LIN {X 0,Y 195.72,Z 619.6,A -85,B 0,C 180,E1 -21671.148,E2 -21671.148} C_VEL
LIN {X 0,Y 194.07,Z 621.131,A -85,B 0,C 180,E1 -21673.162,E2 -21673.162} C_VEL
LIN {X 0,Y 191.846,Z 622.993,A -85,B 0,C 180,E1 -21677.306,E2 -21677.306} C_VEL
LIN {X 0,Y 190.603,Z 623.34,A -85,B 0,C 180,E1 -21681.521,E2 -21681.521} C_VEL
LIN {X 0,Y 190.275,Z 622.063,A -85,B 0,C 180,E1 -21685.766,E2 -21685.766} C_VEL
LIN {X 0,Y 190.318,Z 624.415,A -85,B 0,C 180,E1 -21690.003,E2 -21690.003} C_VEL
LIN {X 0,Y 190.137,Z 625.21,A -85,B 0,C 180,E1 -21693.626,E2 -21693.626} C_VEL
LIN {X 0,Y 190.28,Z 625.058,A -85,B 0,C 180,E1 -21696.364,E2 -21696.364} C_VEL
LIN {X 0,Y 191.05,Z 623.452,A -85,B 0,C 180,E1 -21700.601,E2 -21700.601} C_VEL
LIN {X 0,Y 192.667,Z 620.281,A -85,B 0,C 180,E1 -21704.797,E2 -21704.797} C_VEL
LIN {X 0,Y 194.637,Z 616.754,A -85,B 0,C 180,E1 -21707.876,E2 -21707.876} C_VEL
LIN {X 0,Y 197.217,Z 612.163,A -85,B 0,C 180,E1 -21710.879,E2 -21710.879} C_VEL
LIN {X 0,Y 200.069,Z 606.398,A -85,B 0,C 180,E1 -21713.83,E2 -21713.83} C_VEL
LIN {X 0,Y 203.568,Z 599.221,A -85,B 0,C 180,E1 -21716.67,E2 -21716.67} C_VEL
LIN {X 0,Y 207.615,Z 590.37,A -85,B 0,C 180,E1 -21719.398,E2 -21719.398} C_VEL
LIN {X 0,Y 211.864,Z 580.374,A -85,B 0,C 180,E1 -21721.779,E2 -21721.779} C_VEL
LIN {X 0,Y 215.55,Z 570.262,A -85,B 0,C 180,E1 -21723.664,E2 -21723.664} C_VEL
LIN {X 0,Y 219.069,Z 559.169,A -85,B 0,C 180,E1 -21725.275,E2 -21725.275} C_VEL
LIN {X 0,Y 222.34,Z 546.821,A -85,B 0,C 180,E1 -21726.631,E2 -21726.631} C_VEL
LIN {X 0,Y 225.036,Z 534.261,A -85,B 0,C 180,E1 -21727.59,E2 -21727.59} C_VEL
LIN {X 0,Y 227.03,Z 520.28,A -85,B 0,C 180,E1 -21728.346,E2 -21728.346} C_VEL
LIN {X 0,Y 230.459,Z 474.286,A -85,B 0,C 180,E1 -21729.931,E2 -21729.931} C_VEL
LIN {X 0,Y 230.155,Z 471.556,A -85,B 0,C 180,E1 -21730.175,E2 -21730.175} C_VEL
LIN {X 0,Y 225.508,Z 459.907,A -85,B 0,C 180,E1 -21732.317,E2 -21732.317} C_VEL
LIN {X 0,Y 220.788,Z 450.089,A -85,B 0,C 180,E1 -21734.626,E2 -21734.626} C_VEL
LIN {X 0,Y 216.678,Z 442.974,A -85,B 0,C 180,E1 -21736.78,E2 -21736.78} C_VEL
LIN {X 0,Y 214.755,Z 439.559,A -85,B 0,C 180,E1 -21737.912,E2 -21737.912} C_VEL
LIN {X 0,Y 211.682,Z 434.637,A -85,B 0,C 180,E1 -21739.814,E2 -21739.814} C_VEL
LIN {X 0,Y 208.202,Z 429.263,A -85,B 0,C 180,E1 -21742.258,E2 -21742.258} C_VEL
LIN {X 0,Y 204.808,Z 424.304,A -85,B 0,C 180,E1 -21745.032,E2 -21745.032} C_VEL
LIN {X 0,Y 203.656,Z 422.908,A -85,B 0,C 180,E1 -21746.097,E2 -21746.097} C_VEL
LIN {X 0,Y 199.168,Z 416.55,A -85,B 0,C 180,E1 -21751.575,E2 -21751.575} C_VEL
LIN {X 0,Y 196.529,Z 413.751,A -85,B 0,C 180,E1 -21757.393,E2 -21757.393} C_VEL
LIN {X 0,Y 196.055,Z 412.817,A -85,B 0,C 180,E1 -21761.178,E2 -21761.178} C_VEL
LIN {X 0,Y 196.746,Z 413.155,A -85,B 0,C 180,E1 -21765.52,E2 -21765.52} C_VEL
LIN {X 0,Y 198.963,Z 414.697,A -85,B 0,C 180,E1 -21770.26,E2 -21770.26} C_VEL
LIN {X 0,Y 201.05,Z 417.885,A -85,B 0,C 180,E1 -21773.351,E2 -21773.351} C_VEL
LIN {X 0,Y 204.042,Z 420.336,A -85,B 0,C 180,E1 -21776.378,E2 -21776.378} C_VEL
LIN {X 0,Y 206.331,Z 423.47,A -85,B 0,C 180,E1 -21778.445,E2 -21778.445} C_VEL
LIN {X 0,Y 208.258,Z 425.675,A -85,B 0,C 180,E1 -21779.91,E2 -21779.91} C_VEL
LIN {X 0,Y 211.756,Z 430.682,A -85,B 0,C 180,E1 -21782.378,E2 -21782.378} C_VEL
LIN {X 0,Y 215.572,Z 436.324,A -85,B 0,C 180,E1 -21784.701,E2 -21784.701} C_VEL
LIN {X 0,Y 220.508,Z 444.441,A -85,B 0,C 180,E1 -21787.367,E2 -21787.367} C_VEL
LIN {X 0,Y 225.524,Z 453.78,A -85,B 0,C 180,E1 -21789.803,E2 -21789.803} C_VEL
LIN {X 0,Y 229.635,Z 462.77,A -85,B 0,C 180,E1 -21791.651,E2 -21791.651} C_VEL
LIN {X 0,Y 231.003,Z 466.08,A -85,B 0,C 180,E1 -21792.254,E2 -21792.254} C_VEL
LIN {X 0,Y 227.309,Z 513.393,A -85,B 0,C 180,E1 -21793.884,E2 -21793.884} C_VEL
LIN {X 0,Y 225.489,Z 526.303,A -85,B 0,C 180,E1 -21794.616,E2 -21794.616} C_VEL
LIN {X 0,Y 223.106,Z 538.646,A -85,B 0,C 180,E1 -21795.645,E2 -21795.645} C_VEL
LIN {X 0,Y 220.057,Z 550.738,A -85,B 0,C 180,E1 -21797.031,E2 -21797.031} C_VEL
LIN {X 0,Y 216.86,Z 561.12,A -85,B 0,C 180,E1 -21798.567,E2 -21798.567} C_VEL
LIN {X 0,Y 213.017,Z 571.787,A -85,B 0,C 180,E1 -21800.579,E2 -21800.579} C_VEL
LIN {X 0,Y 208.985,Z 581.554,A -85,B 0,C 180,E1 -21802.981,E2 -21802.981} C_VEL
LIN {X 0,Y 204.885,Z 590.415,A -85,B 0,C 180,E1 -21805.78,E2 -21805.78} C_VEL
LIN {X 0,Y 201.513,Z 596.904,A -85,B 0,C 180,E1 -21808.382,E2 -21808.382} C_VEL
LIN {X 0,Y 198.132,Z 603.112,A -85,B 0,C 180,E1 -21811.641,E2 -21811.641} C_VEL
LIN {X 0,Y 195.241,Z 608.052,A -85,B 0,C 180,E1 -21815.166,E2 -21815.166} C_VEL
LIN {X 0,Y 193.362,Z 611.071,A -85,B 0,C 180,E1 -21818.162,E2 -21818.162} C_VEL
LIN {X 0,Y 191.904,Z 613.201,A -85,B 0,C 180,E1 -21821.24,E2 -21821.24} C_VEL
LIN {X 0,Y 190.5,Z 614.691,A -85,B 0,C 180,E1 -21825.493,E2 -21825.493} C_VEL
LIN {X 0,Y 189.985,Z 614.771,A -85,B 0,C 180,E1 -21828.248,E2 -21828.248} C_VEL
LIN {X 0,Y 189.755,Z 614.193,A -85,B 0,C 180,E1 -21831.059,E2 -21831.059} C_VEL
LIN {X 0,Y 189.779,Z 612.447,A -85,B 0,C 180,E1 -21834.56,E2 -21834.56} C_VEL
LIN {X 0,Y 190.323,Z 609.463,A -85,B 0,C 180,E1 -21838.138,E2 -21838.138} C_VEL
LIN {X 0,Y 191.202,Z 604.893,A -85,B 0,C 180,E1 -21841.906,E2 -21841.906} C_VEL
LIN {X 0,Y 192.232,Z 599.97,A -85,B 0,C 180,E1 -21844.948,E2 -21844.948} C_VEL
LIN {X 0,Y 193.763,Z 593.339,A -85,B 0,C 180,E1 -21848.172,E2 -21848.172} C_VEL
LIN {X 0,Y 195.561,Z 585.609,A -85,B 0,C 180,E1 -21851.126,E2 -21851.126} C_VEL
LIN {X 0,Y 197.618,Z 576.917,A -85,B 0,C 180,E1 -21853.785,E2 -21853.785} C_VEL
LIN {X 0,Y 199.933,Z 566.816,A -85,B 0,C 180,E1 -21856.255,E2 -21856.255} C_VEL
LIN {X 0,Y 201.923,Z 556.858,A -85,B 0,C 180,E1 -21858.198,E2 -21858.198} C_VEL
LIN {X 0,Y 204.183,Z 544.37,A -85,B 0,C 180,E1 -21860.088,E2 -21860.088} C_VEL
LIN {X 0,Y 205.884,Z 532.609,A -85,B 0,C 180,E1 -21861.445,E2 -21861.445} C_VEL
LIN {X 0,Y 207.28,Z 519.795,A -85,B 0,C 180,E1 -21862.512,E2 -21862.512} C_VEL
LIN {X 0,Y 208.32,Z 506.638,A -85,B 0,C 180,E1 -21863.215,E2 -21863.215} C_VEL
LIN {X 0,Y 211.141,Z 450.661,A -85,B 0,C 180,E1 -21865.247,E2 -21865.247} C_VEL
LIN {X 0,Y 202.81,Z 427.829,A -85,B 0,C 180,E1 -21867.418,E2 -21867.418} C_VEL
LIN {X 0,Y 193.596,Z 408.295,A -85,B 0,C 180,E1 -21869.803,E2 -21869.803} C_VEL
LIN {X 0,Y 193.445,Z 407.387,A -85,B 0,C 180,E1 -21869.932,E2 -21869.932} C_VEL
LIN {X 0,Y 192.983,Z 407.442,A -85,B 0,C 180,E1 -21874.174,E2 -21874.174} C_VEL
LIN {X 0,Y 193.081,Z 407.431,A -85,B 0,C 180,E1 -21878.369,E2 -21878.369} C_VEL
LIN {X 0,Y 192.854,Z 407.455,A -85,B 0,C 180,E1 -21882.627,E2 -21882.627} C_VEL
LIN {X 0,Y 192.758,Z 407.473,A -85,B 0,C 180,E1 -21886.956,E2 -21886.956} C_VEL
LIN {X 0,Y 192.636,Z 407.485,A -85,B 0,C 180,E1 -21891.394,E2 -21891.394} C_VEL
LIN {X 0,Y 192.663,Z 407.484,A -85,B 0,C 180,E1 -21894.222,E2 -21894.222} C_VEL
LIN {X 0,Y 192.642,Z 407.476,A -85,B 0,C 180,E1 -21898.886,E2 -21898.886} C_VEL
LIN {X 0,Y 192.59,Z 407.495,A -85,B 0,C 180,E1 -21904.442,E2 -21904.442} C_VEL
LIN {X 0,Y 192.647,Z 407.577,A -85,B 0,C 180,E1 -21905.627,E2 -21905.627} C_VEL
LIN {X 0,Y 200.514,Z 429.954,A -85,B 0,C 180,E1 -21907.562,E2 -21907.562} C_VEL
LIN {X 0,Y 204.611,Z 443.484,A -85,B 0,C 180,E1 -21908.602,E2 -21908.602} C_VEL
LIN {X 0,Y 200.833,Z 511.211,A -85,B 0,C 180,E1 -21911.922,E2 -21911.922} C_VEL
LIN {X 0,Y 199.882,Z 524.754,A -85,B 0,C 180,E1 -21912.963,E2 -21912.963} C_VEL
LIN {X 0,Y 198.418,Z 539.046,A -85,B 0,C 180,E1 -21914.534,E2 -21914.534} C_VEL
LIN {X 0,Y 196.966,Z 550.809,A -85,B 0,C 180,E1 -21916.264,E2 -21916.264} C_VEL
LIN {X 0,Y 195.299,Z 563.165,A -85,B 0,C 180,E1 -21918.585,E2 -21918.585} C_VEL
LIN {X 0,Y 193.693,Z 574.251,A -85,B 0,C 180,E1 -21921.251,E2 -21921.251} C_VEL
LIN {X 0,Y 192.55,Z 582.821,A -85,B 0,C 180,E1 -21923.791,E2 -21923.791} C_VEL
LIN {X 0,Y 191.558,Z 590.579,A -85,B 0,C 180,E1 -21926.61,E2 -21926.61} C_VEL
LIN {X 0,Y 190.673,Z 598.346,A -85,B 0,C 180,E1 -21930.159,E2 -21930.159} C_VEL
LIN {X 0,Y 190.126,Z 604.251,A -85,B 0,C 180,E1 -21933.667,E2 -21933.667} C_VEL
LIN {X 0,Y 189.785,Z 608.454,A -85,B 0,C 180,E1 -21936.992,E2 -21936.992} C_VEL
LIN {X 0,Y 189.845,Z 611.673,A -85,B 0,C 180,E1 -21940.538,E2 -21940.538} C_VEL
LIN {X 0,Y 190.37,Z 613.55,A -85,B 0,C 180,E1 -21943.699,E2 -21943.699} C_VEL
LIN {X 0,Y 191.399,Z 614.57,A -85,B 0,C 180,E1 -21947.272,E2 -21947.272} C_VEL
LIN {X 0,Y 192.6,Z 614.58,A -85,B 0,C 180,E1 -21950.122,E2 -21950.122} C_VEL
LIN {X 0,Y 194.924,Z 613.442,A -85,B 0,C 180,E1 -21953.79,E2 -21953.79} C_VEL
LIN {X 0,Y 197.152,Z 611.798,A -85,B 0,C 180,E1 -21956.445,E2 -21956.445} C_VEL
LIN {X 0,Y 200.801,Z 608.327,A -85,B 0,C 180,E1 -21960,E2 -21960} C_VEL
LIN {X 0,Y 205.018,Z 603.713,A -85,B 0,C 180,E1 -21963.203,E2 -21963.203} C_VEL
LIN {X 0,Y 209.825,Z 597.699,A -85,B 0,C 180,E1 -21966.249,E2 -21966.249} C_VEL
LIN {X 0,Y 214.647,Z 590.895,A -85,B 0,C 180,E1 -21968.853,E2 -21968.853} C_VEL
LIN {X 0,Y 220.368,Z 581.806,A -85,B 0,C 180,E1 -21971.497,E2 -21971.497} C_VEL
LIN {X 0,Y 225.068,Z 573.343,A -85,B 0,C 180,E1 -21973.423,E2 -21973.423} C_VEL
LIN {X 0,Y 230.657,Z 561.717,A -85,B 0,C 180,E1 -21975.462,E2 -21975.462} C_VEL
LIN {X 0,Y 235.084,Z 550.754,A -85,B 0,C 180,E1 -21976.939,E2 -21976.939} C_VEL
LIN {X 0,Y 239.295,Z 538.245,A -85,B 0,C 180,E1 -21978.24,E2 -21978.24} C_VEL
LIN {X 0,Y 242.468,Z 526.564,A -85,B 0,C 180,E1 -21979.141,E2 -21979.141} C_VEL
LIN {X 0,Y 245.063,Z 513.73,A -85,B 0,C 180,E1 -21979.856,E2 -21979.856} C_VEL
LIN {X 0,Y 249.279,Z 484.945,A -85,B 0,C 180,E1 -21981.013,E2 -21981.013} C_VEL
LIN {X 0,Y 249.307,Z 482.556,A -85,B 0,C 180,E1 -21981.299,E2 -21981.299} C_VEL
LIN {X 0,Y 248.726,Z 480.497,A -85,B 0,C 180,E1 -21981.926,E2 -21981.926} C_VEL
LIN {X 0,Y 247.718,Z 479.21,A -85,B 0,C 180,E1 -21982.755,E2 -21982.755} C_VEL
LIN {X 0,Y 244.844,Z 477.488,A -85,B 0,C 180,E1 -21985.136,E2 -21985.136} C_VEL
LIN {X 0,Y 244.529,Z 477.081,A -85,B 0,C 180,E1 -21985.474,E2 -21985.474} C_VEL
LIN {X 0,Y 243.393,Z 474.587,A -85,B 0,C 180,E1 -21987.16,E2 -21987.16} C_VEL
LIN {X 0,Y 242.23,Z 471.931,A -85,B 0,C 180,E1 -21989.553,E2 -21989.553} C_VEL
LIN {X 0,Y 241.395,Z 470.813,A -85,B 0,C 180,E1 -21992.407,E2 -21992.407} C_VEL
LIN {X 0,Y 241.409,Z 470.899,A -85,B 0,C 180,E1 -21995.609,E2 -21995.609} C_VEL
LIN {X 0,Y 242.353,Z 472.652,A -85,B 0,C 180,E1 -21998.736,E2 -21998.736} C_VEL
LIN {X 0,Y 243.872,Z 476.256,A -85,B 0,C 180,E1 -22001.516,E2 -22001.516} C_VEL
LIN {X 0,Y 245.796,Z 480.734,A -85,B 0,C 180,E1 -22003.961,E2 -22003.961} C_VEL
LIN {X 0,Y 246.892,Z 483.497,A -85,B 0,C 180,E1 -22005.123,E2 -22005.123} C_VEL
LIN {X 0,Y 240.741,Z 522.488,A -85,B 0,C 180,E1 -22006.758,E2 -22006.758} C_VEL
LIN {X 0,Y 237.486,Z 536.119,A -85,B 0,C 180,E1 -22007.542,E2 -22007.542} C_VEL
LIN {X 0,Y 233.407,Z 548.738,A -85,B 0,C 180,E1 -22008.518,E2 -22008.518} C_VEL
LIN {X 0,Y 228.53,Z 560.939,A -85,B 0,C 180,E1 -22009.777,E2 -22009.777} C_VEL
LIN {X 0,Y 222.432,Z 573.961,A -85,B 0,C 180,E1 -22011.682,E2 -22011.682} C_VEL
LIN {X 0,Y 217.63,Z 582.71,A -85,B 0,C 180,E1 -22013.318,E2 -22013.318} C_VEL
LIN {X 0,Y 211.65,Z 592.278,A -85,B 0,C 180,E1 -22015.636,E2 -22015.636} C_VEL
LIN {X 0,Y 206.176,Z 600.165,A -85,B 0,C 180,E1 -22018.109,E2 -22018.109} C_VEL
LIN {X 0,Y 200.984,Z 607.02,A -85,B 0,C 180,E1 -22020.95,E2 -22020.95} C_VEL
LIN {X 0,Y 196.912,Z 611.796,A -85,B 0,C 180,E1 -22023.507,E2 -22023.507} C_VEL
LIN {X 0,Y 193.283,Z 615.915,A -85,B 0,C 180,E1 -22026.427,E2 -22026.427} C_VEL
LIN {X 0,Y 191.042,Z 618.136,A -85,B 0,C 180,E1 -22028.418,E2 -22028.418} C_VEL
LIN {X 0,Y 187.282,Z 621.302,A -85,B 0,C 180,E1 -22032.533,E2 -22032.533} C_VEL
LIN {X 0,Y 184.903,Z 622.943,A -85,B 0,C 180,E1 -22036.82,E2 -22036.82} C_VEL
LIN {X 0,Y 183.563,Z 622.993,A -85,B 0,C 180,E1 -22041.194,E2 -22041.194} C_VEL
LIN {X 0,Y 183.201,Z 621.563,A -85,B 0,C 180,E1 -22045.722,E2 -22045.722} C_VEL
LIN {X 0,Y 183.116,Z 623.011,A -85,B 0,C 180,E1 -22047.803,E2 -22047.803} C_VEL
LIN {X 0,Y 183.22,Z 624.102,A -85,B 0,C 180,E1 -22050.003,E2 -22050.003} C_VEL
LIN {X 0,Y 183.054,Z 624.966,A -85,B 0,C 180,E1 -22053.417,E2 -22053.417} C_VEL
LIN {X 0,Y 183.213,Z 624.889,A -85,B 0,C 180,E1 -22056.611,E2 -22056.611} C_VEL
LIN {X 0,Y 183.517,Z 624.357,A -85,B 0,C 180,E1 -22058.814,E2 -22058.814} C_VEL
LIN {X 0,Y 184.817,Z 622.081,A -85,B 0,C 180,E1 -22063.192,E2 -22063.192} C_VEL
LIN {X 0,Y 186.415,Z 619.31,A -85,B 0,C 180,E1 -22066.428,E2 -22066.428} C_VEL
LIN {X 0,Y 188.727,Z 615.542,A -85,B 0,C 180,E1 -22069.585,E2 -22069.585} C_VEL
LIN {X 0,Y 191.568,Z 610.685,A -85,B 0,C 180,E1 -22072.659,E2 -22072.659} C_VEL
LIN {X 0,Y 195.358,Z 603.525,A -85,B 0,C 180,E1 -22076.151,E2 -22076.151} C_VEL
LIN {X 0,Y 199.338,Z 595.77,A -85,B 0,C 180,E1 -22079.001,E2 -22079.001} C_VEL
LIN {X 0,Y 203.05,Z 587.911,A -85,B 0,C 180,E1 -22081.28,E2 -22081.28} C_VEL
LIN {X 0,Y 207.593,Z 577.326,A -85,B 0,C 180,E1 -22083.67,E2 -22083.67} C_VEL
LIN {X 0,Y 211.547,Z 566.614,A -85,B 0,C 180,E1 -22085.551,E2 -22085.551} C_VEL
LIN {X 0,Y 215.332,Z 554.54,A -85,B 0,C 180,E1 -22087.145,E2 -22087.145} C_VEL
LIN {X 0,Y 218.326,Z 542.986,A -85,B 0,C 180,E1 -22088.294,E2 -22088.294} C_VEL
LIN {X 0,Y 220.995,Z 529.936,A -85,B 0,C 180,E1 -22089.205,E2 -22089.205} C_VEL
LIN {X 0,Y 222.7,Z 516.089,A -85,B 0,C 180,E1 -22089.872,E2 -22089.872} C_VEL
LIN {X 0,Y 225.877,Z 475.392,A -85,B 0,C 180,E1 -22091.274,E2 -22091.274} C_VEL
LIN {X 0,Y 222.659,Z 466.731,A -85,B 0,C 180,E1 -22092.857,E2 -22092.857} C_VEL
LIN {X 0,Y 218.886,Z 458.171,A -85,B 0,C 180,E1 -22094.81,E2 -22094.81} C_VEL
LIN {X 0,Y 214.768,Z 450.261,A -85,B 0,C 180,E1 -22097.072,E2 -22097.072} C_VEL
LIN {X 0,Y 211.767,Z 444.948,A -85,B 0,C 180,E1 -22098.91,E2 -22098.91} C_VEL
LIN {X 0,Y 209.193,Z 440.674,A -85,B 0,C 180,E1 -22100.6,E2 -22100.6} C_VEL
LIN {X 0,Y 205.948,Z 435.399,A -85,B 0,C 180,E1 -22103.058,E2 -22103.058} C_VEL
LIN {X 0,Y 202.382,Z 429.965,A -85,B 0,C 180,E1 -22106.246,E2 -22106.246} C_VEL
LIN {X 0,Y 197.854,Z 423.395,A -85,B 0,C 180,E1 -22111.935,E2 -22111.935} C_VEL
LIN {X 0,Y 195.378,Z 420.67,A -85,B 0,C 180,E1 -22117.809,E2 -22117.809} C_VEL
LIN {X 0,Y 195.019,Z 419.868,A -85,B 0,C 180,E1 -22121.075,E2 -22121.075} C_VEL
LIN {X 0,Y 195.667,Z 420.166,A -85,B 0,C 180,E1 -22125.438,E2 -22125.438} C_VEL
LIN {X 0,Y 197.663,Z 421.666,A -85,B 0,C 180,E1 -22129.925,E2 -22129.925} C_VEL
LIN {X 0,Y 199.777,Z 424.81,A -85,B 0,C 180,E1 -22133.118,E2 -22133.118} C_VEL
LIN {X 0,Y 202.528,Z 427.29,A -85,B 0,C 180,E1 -22136.02,E2 -22136.02} C_VEL
LIN {X 0,Y 204.674,Z 430.212,A -85,B 0,C 180,E1 -22138.032,E2 -22138.032} C_VEL
LIN {X 0,Y 206.217,Z 432.116,A -85,B 0,C 180,E1 -22139.268,E2 -22139.268} C_VEL
LIN {X 0,Y 210.405,Z 438.444,A -85,B 0,C 180,E1 -22142.342,E2 -22142.342} C_VEL
LIN {X 0,Y 213.122,Z 442.572,A -85,B 0,C 180,E1 -22144.044,E2 -22144.044} C_VEL
LIN {X 0,Y 217.554,Z 450.264,A -85,B 0,C 180,E1 -22146.598,E2 -22146.598} C_VEL
LIN {X 0,Y 222.038,Z 458.885,A -85,B 0,C 180,E1 -22148.908,E2 -22148.908} C_VEL
LIN {X 0,Y 225.885,Z 467.674,A -85,B 0,C 180,E1 -22150.759,E2 -22150.759} C_VEL
LIN {X 0,Y 226.279,Z 468.651,A -85,B 0,C 180,E1 -22150.944,E2 -22150.944} C_VEL
LIN {X 0,Y 222.592,Z 513.888,A -85,B 0,C 180,E1 -22152.537,E2 -22152.537} C_VEL
LIN {X 0,Y 220.629,Z 527.039,A -85,B 0,C 180,E1 -22153.3,E2 -22153.3} C_VEL
LIN {X 0,Y 218.1,Z 539.38,A -85,B 0,C 180,E1 -22154.36,E2 -22154.36} C_VEL
LIN {X 0,Y 214.947,Z 551.16,A -85,B 0,C 180,E1 -22155.734,E2 -22155.734} C_VEL
LIN {X 0,Y 211.331,Z 562.279,A -85,B 0,C 180,E1 -22157.416,E2 -22157.416} C_VEL
LIN {X 0,Y 207.656,Z 571.974,A -85,B 0,C 180,E1 -22159.29,E2 -22159.29} C_VEL
LIN {X 0,Y 203.87,Z 580.756,A -85,B 0,C 180,E1 -22161.439,E2 -22161.439} C_VEL
LIN {X 0,Y 199.436,Z 589.861,A -85,B 0,C 180,E1 -22164.303,E2 -22164.303} C_VEL
LIN {X 0,Y 195.34,Z 597.352,A -85,B 0,C 180,E1 -22167.354,E2 -22167.354} C_VEL
LIN {X 0,Y 191.526,Z 603.807,A -85,B 0,C 180,E1 -22170.913,E2 -22170.913} C_VEL
LIN {X 0,Y 188.954,Z 607.901,A -85,B 0,C 180,E1 -22173.912,E2 -22173.912} C_VEL
LIN {X 0,Y 186.464,Z 611.57,A -85,B 0,C 180,E1 -22177.669,E2 -22177.669} C_VEL
LIN {X 0,Y 185.053,Z 613.449,A -85,B 0,C 180,E1 -22180.57,E2 -22180.57} C_VEL
LIN {X 0,Y 183.974,Z 614.608,A -85,B 0,C 180,E1 -22183.459,E2 -22183.459} C_VEL
LIN {X 0,Y 183.118,Z 615.045,A -85,B 0,C 180,E1 -22186.821,E2 -22186.821} C_VEL
LIN {X 0,Y 182.676,Z 614.523,A -85,B 0,C 180,E1 -22190.305,E2 -22190.305} C_VEL
LIN {X 0,Y 182.65,Z 612.938,A -85,B 0,C 180,E1 -22193.905,E2 -22193.905} C_VEL
LIN {X 0,Y 183.127,Z 610.142,A -85,B 0,C 180,E1 -22197.599,E2 -22197.599} C_VEL
LIN {X 0,Y 183.983,Z 605.786,A -85,B 0,C 180,E1 -22201.473,E2 -22201.473} C_VEL
LIN {X 0,Y 185.24,Z 599.853,A -85,B 0,C 180,E1 -22205.33,E2 -22205.33} C_VEL
LIN {X 0,Y 186.949,Z 592.733,A -85,B 0,C 180,E1 -22208.832,E2 -22208.832} C_VEL
LIN {X 0,Y 189.024,Z 584.112,A -85,B 0,C 180,E1 -22212.134,E2 -22212.134} C_VEL
LIN {X 0,Y 191.037,Z 575.886,A -85,B 0,C 180,E1 -22214.646,E2 -22214.646} C_VEL
LIN {X 0,Y 193.444,Z 565.663,A -85,B 0,C 180,E1 -22217.14,E2 -22217.14} C_VEL
LIN {X 0,Y 195.832,Z 553.864,A -85,B 0,C 180,E1 -22219.399,E2 -22219.399} C_VEL
LIN {X 0,Y 197.9,Z 542.431,A -85,B 0,C 180,E1 -22221.086,E2 -22221.086} C_VEL
LIN {X 0,Y 199.76,Z 529.153,A -85,B 0,C 180,E1 -22222.543,E2 -22222.543} C_VEL
LIN {X 0,Y 201.13,Z 516.229,A -85,B 0,C 180,E1 -22223.54,E2 -22223.54} C_VEL
LIN {X 0,Y 202.134,Z 501.041,A -85,B 0,C 180,E1 -22224.239,E2 -22224.239} C_VEL
LIN {X 0,Y 204.656,Z 452.16,A -85,B 0,C 180,E1 -22226.059,E2 -22226.059} C_VEL
LIN {X 0,Y 196.883,Z 430.644,A -85,B 0,C 180,E1 -22228.2,E2 -22228.2} C_VEL
LIN {X 0,Y 187.869,Z 411.874,A -85,B 0,C 180,E1 -22230.62,E2 -22230.62} C_VEL
LIN {X 0,Y 186.468,Z 409.162,A -85,B 0,C 180,E1 -22231.009,E2 -22231.009} C_VEL
LIN {X 0,Y 186.288,Z 408.284,A -85,B 0,C 180,E1 -22231.145,E2 -22231.145} C_VEL
LIN {X 0,Y 186.031,Z 408.312,A -85,B 0,C 180,E1 -22238.689,E2 -22238.689} C_VEL
LIN {X 0,Y 185.766,Z 408.338,A -85,B 0,C 180,E1 -22243.117,E2 -22243.117} C_VEL
LIN {X 0,Y 185.69,Z 408.349,A -85,B 0,C 180,E1 -22247.622,E2 -22247.622} C_VEL
LIN {X 0,Y 185.596,Z 408.367,A -85,B 0,C 180,E1 -22252.248,E2 -22252.248} C_VEL
LIN {X 0,Y 185.558,Z 408.353,A -85,B 0,C 180,E1 -22257.029,E2 -22257.029} C_VEL
LIN {X 0,Y 185.575,Z 408.357,A -85,B 0,C 180,E1 -22259.49,E2 -22259.49} C_VEL
LIN {X 0,Y 185.568,Z 408.369,A -85,B 0,C 180,E1 -22264.944,E2 -22264.944} C_VEL
LIN {X 0,Y 193.936,Z 432.102,A -85,B 0,C 180,E1 -22267.116,E2 -22267.116} C_VEL
LIN {X 0,Y 197.668,Z 444.58,A -85,B 0,C 180,E1 -22268.114,E2 -22268.114} C_VEL
LIN {X 0,Y 193.894,Z 511.321,A -85,B 0,C 180,E1 -22271.52,E2 -22271.52} C_VEL
LIN {X 0,Y 193.005,Z 523.779,A -85,B 0,C 180,E1 -22272.491,E2 -22272.491} C_VEL
LIN {X 0,Y 191.681,Z 536.813,A -85,B 0,C 180,E1 -22273.921,E2 -22273.921} C_VEL
LIN {X 0,Y 190.13,Z 549.47,A -85,B 0,C 180,E1 -22275.757,E2 -22275.757} C_VEL
LIN {X 0,Y 188.605,Z 560.762,A -85,B 0,C 180,E1 -22277.876,E2 -22277.876} C_VEL
LIN {X 0,Y 187.067,Z 571.191,A -85,B 0,C 180,E1 -22280.306,E2 -22280.306} C_VEL
LIN {X 0,Y 185.815,Z 579.758,A -85,B 0,C 180,E1 -22282.759,E2 -22282.759} C_VEL
LIN {X 0,Y 184.702,Z 588.168,A -85,B 0,C 180,E1 -22285.725,E2 -22285.725} C_VEL
LIN {X 0,Y 183.82,Z 595.508,A -85,B 0,C 180,E1 -22288.926,E2 -22288.926} C_VEL
LIN {X 0,Y 183.333,Z 600.917,A -85,B 0,C 180,E1 -22291.841,E2 -22291.841} C_VEL
LIN {X 0,Y 182.866,Z 605.595,A -85,B 0,C 180,E1 -22294.991,E2 -22294.991} C_VEL
LIN {X 0,Y 182.685,Z 609.658,A -85,B 0,C 180,E1 -22298.577,E2 -22298.577} C_VEL
LIN {X 0,Y 182.938,Z 612.464,A -85,B 0,C 180,E1 -22302.101,E2 -22302.101} C_VEL
LIN {X 0,Y 183.426,Z 613.712,A -85,B 0,C 180,E1 -22304.442,E2 -22304.442} C_VEL
LIN {X 0,Y 184.067,Z 614.506,A -85,B 0,C 180,E1 -22306.756,E2 -22306.756} C_VEL
LIN {X 0,Y 185.463,Z 614.885,A -85,B 0,C 180,E1 -22310.128,E2 -22310.128} C_VEL
LIN {X 0,Y 187.522,Z 614.276,A -85,B 0,C 180,E1 -22313.544,E2 -22313.544} C_VEL
LIN {X 0,Y 190.065,Z 612.795,A -85,B 0,C 180,E1 -22316.676,E2 -22316.676} C_VEL
LIN {X 0,Y 193.425,Z 610.128,A -85,B 0,C 180,E1 -22320,E2 -22320} C_VEL
LIN {X 0,Y 197.023,Z 606.736,A -85,B 0,C 180,E1 -22322.884,E2 -22322.884} C_VEL
LIN {X 0,Y 201.792,Z 601.674,A -85,B 0,C 180,E1 -22325.997,E2 -22325.997} C_VEL
LIN {X 0,Y 206.702,Z 595.648,A -85,B 0,C 180,E1 -22328.773,E2 -22328.773} C_VEL
LIN {X 0,Y 212.355,Z 587.929,A -85,B 0,C 180,E1 -22331.453,E2 -22331.453} C_VEL
LIN {X 0,Y 218.267,Z 578.607,A -85,B 0,C 180,E1 -22333.937,E2 -22333.937} C_VEL
LIN {X 0,Y 223.827,Z 568.571,A -85,B 0,C 180,E1 -22335.947,E2 -22335.947} C_VEL
LIN {X 0,Y 228.969,Z 557.747,A -85,B 0,C 180,E1 -22337.656,E2 -22337.656} C_VEL
LIN {X 0,Y 233.721,Z 545.754,A -85,B 0,C 180,E1 -22339.099,E2 -22339.099} C_VEL
LIN {X 0,Y 238.001,Z 532.294,A -85,B 0,C 180,E1 -22340.302,E2 -22340.302} C_VEL
LIN {X 0,Y 241.53,Z 517.671,A -85,B 0,C 180,E1 -22341.216,E2 -22341.216} C_VEL
LIN {X 0,Y 246.734,Z 484.983,A -85,B 0,C 180,E1 -22342.551,E2 -22342.551} C_VEL
LIN {X 0,Y 246.958,Z 483.027,A -85,B 0,C 180,E1 -22342.679,E2 -22342.679} C_VEL
LIN {X 0,Y 245.435,Z 479.266,A -85,B 0,C 180,E1 -22344.338,E2 -22344.338} C_VEL
LIN {X 0,Y 244.529,Z 477.081,A -85,B 0,C 180,E1 -22345.474,E2 -22345.474} C_VEL
LIN {X 0,Y 243.399,Z 476.014,A -85,B 0,C 180,E1 -22346.816,E2 -22346.816} C_VEL
LIN {X 0,Y 242.248,Z 476.015,A -85,B 0,C 180,E1 -22348.196,E2 -22348.196} C_VEL
LIN {X 0,Y 240.077,Z 477.675,A -85,B 0,C 180,E1 -22351.973,E2 -22351.973} C_VEL
LIN {X 0,Y 239.872,Z 477.7,A -85,B 0,C 180,E1 -22352.935,E2 -22352.935} C_VEL
LIN {X 0,Y 240.01,Z 478.093,A -85,B 0,C 180,E1 -22356.08,E2 -22356.08} C_VEL
LIN {X 0,Y 240.713,Z 479.367,A -85,B 0,C 180,E1 -22358.334,E2 -22358.334} C_VEL
LIN {X 0,Y 242.003,Z 482.826,A -85,B 0,C 180,E1 -22361.043,E2 -22361.043} C_VEL
LIN {X 0,Y 243.655,Z 486.99,A -85,B 0,C 180,E1 -22363.356,E2 -22363.356} C_VEL
LIN {X 0,Y 243.924,Z 488.048,A -85,B 0,C 180,E1 -22363.749,E2 -22363.749} C_VEL
LIN {X 0,Y 238.424,Z 521.478,A -85,B 0,C 180,E1 -22365.119,E2 -22365.119} C_VEL
LIN {X 0,Y 235.029,Z 535.099,A -85,B 0,C 180,E1 -22365.87,E2 -22365.87} C_VEL
LIN {X 0,Y 230.905,Z 547.469,A -85,B 0,C 180,E1 -22366.782,E2 -22366.782} C_VEL
LIN {X 0,Y 225.857,Z 559.813,A -85,B 0,C 180,E1 -22368.012,E2 -22368.012} C_VEL
LIN {X 0,Y 220.571,Z 570.831,A -85,B 0,C 180,E1 -22369.522,E2 -22369.522} C_VEL
LIN {X 0,Y 214.342,Z 581.763,A -85,B 0,C 180,E1 -22371.469,E2 -22371.469} C_VEL
LIN {X 0,Y 208.005,Z 591.495,A -85,B 0,C 180,E1 -22373.755,E2 -22373.755} C_VEL
LIN {X 0,Y 202.149,Z 599.406,A -85,B 0,C 180,E1 -22376.206,E2 -22376.206} C_VEL
LIN {X 0,Y 196.877,Z 605.88,A -85,B 0,C 180,E1 -22378.831,E2 -22378.831} C_VEL
LIN {X 0,Y 192.002,Z 611.19,A -85,B 0,C 180,E1 -22381.589,E2 -22381.589} C_VEL
LIN {X 0,Y 188.043,Z 615.342,A -85,B 0,C 180,E1 -22384.548,E2 -22384.548} C_VEL
LIN {X 0,Y 184.485,Z 618.568,A -85,B 0,C 180,E1 -22387.611,E2 -22387.611} C_VEL
LIN {X 0,Y 180.523,Z 621.485,A -85,B 0,C 180,E1 -22391.857,E2 -22391.857} C_VEL
LIN {X 0,Y 177.981,Z 622.803,A -85,B 0,C 180,E1 -22396.298,E2 -22396.298} C_VEL
LIN {X 0,Y 176.545,Z 622.635,A -85,B 0,C 180,E1 -22400.841,E2 -22400.841} C_VEL
LIN {X 0,Y 176.138,Z 621.012,A -85,B 0,C 180,E1 -22405.426,E2 -22405.426} C_VEL
LIN {X 0,Y 176.023,Z 622.601,A -85,B 0,C 180,E1 -22407.715,E2 -22407.715} C_VEL
LIN {X 0,Y 176.124,Z 623.774,A -85,B 0,C 180,E1 -22410.003,E2 -22410.003} C_VEL
LIN {X 0,Y 175.971,Z 624.644,A -85,B 0,C 180,E1 -22413.178,E2 -22413.178} C_VEL
LIN {X 0,Y 176.142,Z 624.708,A -85,B 0,C 180,E1 -22416.878,E2 -22416.878} C_VEL
LIN {X 0,Y 176.481,Z 624.25,A -85,B 0,C 180,E1 -22419.169,E2 -22419.169} C_VEL
LIN {X 0,Y 177.066,Z 623.377,A -85,B 0,C 180,E1 -22421.45,E2 -22421.45} C_VEL
LIN {X 0,Y 178.917,Z 620.417,A -85,B 0,C 180,E1 -22425.963,E2 -22425.963} C_VEL
LIN {X 0,Y 181.175,Z 617.099,A -85,B 0,C 180,E1 -22429.255,E2 -22429.255} C_VEL
LIN {X 0,Y 183.995,Z 612.754,A -85,B 0,C 180,E1 -22432.458,E2 -22432.458} C_VEL
LIN {X 0,Y 187.784,Z 606.289,A -85,B 0,C 180,E1 -22436.074,E2 -22436.074} C_VEL
LIN {X 0,Y 191.723,Z 599.201,A -85,B 0,C 180,E1 -22439.062,E2 -22439.062} C_VEL
LIN {X 0,Y 196.214,Z 590.453,A -85,B 0,C 180,E1 -22441.895,E2 -22441.895} C_VEL
LIN {X 0,Y 200.488,Z 581.56,A -85,B 0,C 180,E1 -22444.119,E2 -22444.119} C_VEL
LIN {X 0,Y 204.504,Z 571.905,A -85,B 0,C 180,E1 -22446.055,E2 -22446.055} C_VEL
LIN {X 0,Y 208.31,Z 561.384,A -85,B 0,C 180,E1 -22447.701,E2 -22447.701} C_VEL
LIN {X 0,Y 211.85,Z 549.762,A -85,B 0,C 180,E1 -22449.076,E2 -22449.076} C_VEL
LIN {X 0,Y 214.793,Z 537.91,A -85,B 0,C 180,E1 -22450.106,E2 -22450.106} C_VEL
LIN {X 0,Y 217.24,Z 524.497,A -85,B 0,C 180,E1 -22450.925,E2 -22450.925} C_VEL
LIN {X 0,Y 218.876,Z 507.47,A -85,B 0,C 180,E1 -22451.614,E2 -22451.614} C_VEL
LIN {X 0,Y 221.346,Z 477.75,A -85,B 0,C 180,E1 -22452.621,E2 -22452.621} C_VEL
LIN {X 0,Y 217.326,Z 467.199,A -85,B 0,C 180,E1 -22454.8,E2 -22454.8} C_VEL
LIN {X 0,Y 213.819,Z 459.719,A -85,B 0,C 180,E1 -22456.775,E2 -22456.775} C_VEL
LIN {X 0,Y 209.792,Z 451.786,A -85,B 0,C 180,E1 -22459.325,E2 -22459.325} C_VEL
LIN {X 0,Y 206.719,Z 446.565,A -85,B 0,C 180,E1 -22461.472,E2 -22461.472} C_VEL
LIN {X 0,Y 203.846,Z 441.711,A -85,B 0,C 180,E1 -22463.774,E2 -22463.774} C_VEL
LIN {X 0,Y 200.529,Z 436.382,A -85,B 0,C 180,E1 -22466.969,E2 -22466.969} C_VEL
LIN {X 0,Y 196.543,Z 430.276,A -85,B 0,C 180,E1 -22472.299,E2 -22472.299} C_VEL
LIN {X 0,Y 194.244,Z 427.581,A -85,B 0,C 180,E1 -22478.232,E2 -22478.232} C_VEL
LIN {X 0,Y 193.983,Z 426.919,A -85,B 0,C 180,E1 -22480.97,E2 -22480.97} C_VEL
LIN {X 0,Y 194.592,Z 427.156,A -85,B 0,C 180,E1 -22485.356,E2 -22485.356} C_VEL
LIN {X 0,Y 196.366,Z 428.6,A -85,B 0,C 180,E1 -22489.561,E2 -22489.561} C_VEL
LIN {X 0,Y 198.487,Z 431.752,A -85,B 0,C 180,E1 -22492.862,E2 -22492.862} C_VEL
LIN {X 0,Y 200.825,Z 433.945,A -85,B 0,C 180,E1 -22495.453,E2 -22495.453} C_VEL
LIN {X 0,Y 203.119,Z 437.021,A -85,B 0,C 180,E1 -22497.675,E2 -22497.675} C_VEL
LIN {X 0,Y 204.188,Z 438.572,A -85,B 0,C 180,E1 -22498.613,E2 -22498.613} C_VEL
LIN {X 0,Y 208.166,Z 444.784,A -85,B 0,C 180,E1 -22501.685,E2 -22501.685} C_VEL
LIN {X 0,Y 210.592,Z 448.667,A -85,B 0,C 180,E1 -22503.306,E2 -22503.306} C_VEL
LIN {X 0,Y 215.21,Z 457.057,A -85,B 0,C 180,E1 -22506.119,E2 -22506.119} C_VEL
LIN {X 0,Y 219.303,Z 465.515,A -85,B 0,C 180,E1 -22508.332,E2 -22508.332} C_VEL
LIN {X 0,Y 221.751,Z 471.416,A -85,B 0,C 180,E1 -22509.615,E2 -22509.615} C_VEL
LIN {X 0,Y 218.076,Z 514.012,A -85,B 0,C 180,E1 -22511.111,E2 -22511.111} C_VEL
LIN {X 0,Y 216.062,Z 527.07,A -85,B 0,C 180,E1 -22511.869,E2 -22511.869} C_VEL
LIN {X 0,Y 213.644,Z 538.53,A -85,B 0,C 180,E1 -22512.839,E2 -22512.839} C_VEL
LIN {X 0,Y 210.636,Z 549.617,A -85,B 0,C 180,E1 -22514.083,E2 -22514.083} C_VEL
LIN {X 0,Y 206.831,Z 561.032,A -85,B 0,C 180,E1 -22515.774,E2 -22515.774} C_VEL
LIN {X 0,Y 202.8,Z 571.296,A -85,B 0,C 180,E1 -22517.736,E2 -22517.736} C_VEL
LIN {X 0,Y 198.617,Z 580.501,A -85,B 0,C 180,E1 -22519.97,E2 -22519.97} C_VEL
LIN {X 0,Y 194.37,Z 588.9,A -85,B 0,C 180,E1 -22522.598,E2 -22522.598} C_VEL
LIN {X 0,Y 190.482,Z 595.762,A -85,B 0,C 180,E1 -22525.315,E2 -22525.315} C_VEL
LIN {X 0,Y 186.384,Z 602.4,A -85,B 0,C 180,E1 -22528.75,E2 -22528.75} C_VEL
LIN {X 0,Y 182.715,Z 607.798,A -85,B 0,C 180,E1 -22532.582,E2 -22532.582} C_VEL
LIN {X 0,Y 180.449,Z 610.985,A -85,B 0,C 180,E1 -22535.748,E2 -22535.748} C_VEL
LIN {X 0,Y 178.584,Z 613.287,A -85,B 0,C 180,E1 -22539.026,E2 -22539.026} C_VEL
LIN {X 0,Y 177.182,Z 614.705,A -85,B 0,C 180,E1 -22542.401,E2 -22542.401} C_VEL
LIN {X 0,Y 176.191,Z 615.239,A -85,B 0,C 180,E1 -22545.889,E2 -22545.889} C_VEL
LIN {X 0,Y 175.591,Z 614.659,A -85,B 0,C 180,E1 -22550.175,E2 -22550.175} C_VEL
LIN {X 0,Y 175.522,Z 613.367,A -85,B 0,C 180,E1 -22553.208,E2 -22553.208} C_VEL
LIN {X 0,Y 175.907,Z 610.729,A -85,B 0,C 180,E1 -22557.036,E2 -22557.036} C_VEL
LIN {X 0,Y 176.73,Z 606.628,A -85,B 0,C 180,E1 -22561.03,E2 -22561.03} C_VEL
LIN {X 0,Y 177.697,Z 602.242,A -85,B 0,C 180,E1 -22564.208,E2 -22564.208} C_VEL
LIN {X 0,Y 179.045,Z 596.475,A -85,B 0,C 180,E1 -22567.495,E2 -22567.495} C_VEL
LIN {X 0,Y 180.822,Z 589.363,A -85,B 0,C 180,E1 -22570.706,E2 -22570.706} C_VEL
LIN {X 0,Y 183.005,Z 580.865,A -85,B 0,C 180,E1 -22573.758,E2 -22573.758} C_VEL
LIN {X 0,Y 185.474,Z 570.969,A -85,B 0,C 180,E1 -22576.577,E2 -22576.577} C_VEL
LIN {X 0,Y 187.946,Z 559.997,A -85,B 0,C 180,E1 -22579.017,E2 -22579.017} C_VEL
LIN {X 0,Y 190.204,Z 548.836,A -85,B 0,C 180,E1 -22580.962,E2 -22580.962} C_VEL
LIN {X 0,Y 192.219,Z 536.665,A -85,B 0,C 180,E1 -22582.59,E2 -22582.59} C_VEL
LIN {X 0,Y 193.92,Z 522.967,A -85,B 0,C 180,E1 -22583.919,E2 -22583.919} C_VEL
LIN {X 0,Y 195.234,Z 509.783,A -85,B 0,C 180,E1 -22584.737,E2 -22584.737} C_VEL
LIN {X 0,Y 198.236,Z 453.578,A -85,B 0,C 180,E1 -22586.925,E2 -22586.925} C_VEL
LIN {X 0,Y 190.875,Z 433.359,A -85,B 0,C 180,E1 -22589.039,E2 -22589.039} C_VEL
LIN {X 0,Y 182.601,Z 416.1,A -85,B 0,C 180,E1 -22591.36,E2 -22591.36} C_VEL
LIN {X 0,Y 179.379,Z 410.332,A -85,B 0,C 180,E1 -22592.278,E2 -22592.278} C_VEL
LIN {X 0,Y 179.108,Z 409.17,A -85,B 0,C 180,E1 -22592.457,E2 -22592.457} C_VEL
LIN {X 0,Y 178.98,Z 409.192,A -85,B 0,C 180,E1 -22599.034,E2 -22599.034} C_VEL
LIN {X 0,Y 178.688,Z 409.222,A -85,B 0,C 180,E1 -22603.647,E2 -22603.647} C_VEL
LIN {X 0,Y 178.65,Z 409.221,A -85,B 0,C 180,E1 -22608.34,E2 -22608.34} C_VEL
LIN {X 0,Y 178.51,Z 409.249,A -85,B 0,C 180,E1 -22613.182,E2 -22613.182} C_VEL
LIN {X 0,Y 178.483,Z 409.233,A -85,B 0,C 180,E1 -22618.194,E2 -22618.194} C_VEL
LIN {X 0,Y 178.474,Z 409.249,A -85,B 0,C 180,E1 -22620.788,E2 -22620.788} C_VEL
LIN {X 0,Y 178.515,Z 409.284,A -85,B 0,C 180,E1 -22624.291,E2 -22624.291} C_VEL
LIN {X 0,Y 187.333,Z 434.221,A -85,B 0,C 180,E1 -22626.633,E2 -22626.633} C_VEL
LIN {X 0,Y 190.778,Z 445.645,A -85,B 0,C 180,E1 -22627.597,E2 -22627.597} C_VEL
LIN {X 0,Y 186.946,Z 511.516,A -85,B 0,C 180,E1 -22631.093,E2 -22631.093} C_VEL
LIN {X 0,Y 185.888,Z 525.026,A -85,B 0,C 180,E1 -22632.202,E2 -22632.202} C_VEL
LIN {X 0,Y 184.449,Z 538.717,A -85,B 0,C 180,E1 -22633.815,E2 -22633.815} C_VEL
LIN {X 0,Y 182.82,Z 551.474,A -85,B 0,C 180,E1 -22635.832,E2 -22635.832} C_VEL
LIN {X 0,Y 181.17,Z 563.081,A -85,B 0,C 180,E1 -22638.182,E2 -22638.182} C_VEL
LIN {X 0,Y 179.589,Z 573.584,A -85,B 0,C 180,E1 -22640.873,E2 -22640.873} C_VEL
LIN {X 0,Y 178.333,Z 582.722,A -85,B 0,C 180,E1 -22643.762,E2 -22643.762} C_VEL
LIN {X 0,Y 177.249,Z 590.914,A -85,B 0,C 180,E1 -22646.962,E2 -22646.962} C_VEL
LIN {X 0,Y 176.515,Z 597.49,A -85,B 0,C 180,E1 -22650.154,E2 -22650.154} C_VEL
LIN {X 0,Y 176.119,Z 601.817,A -85,B 0,C 180,E1 -22652.683,E2 -22652.683} C_VEL
LIN {X 0,Y 175.664,Z 606.875,A -85,B 0,C 180,E1 -22656.416,E2 -22656.416} C_VEL
LIN {X 0,Y 175.629,Z 610.567,A -85,B 0,C 180,E1 -22660.114,E2 -22660.114} C_VEL
LIN {X 0,Y 176.171,Z 613.124,A -85,B 0,C 180,E1 -22663.784,E2 -22663.784} C_VEL
LIN {X 0,Y 176.753,Z 614.236,A -85,B 0,C 180,E1 -22666.198,E2 -22666.198} C_VEL
LIN {X 0,Y 178.31,Z 615.111,A -85,B 0,C 180,E1 -22670.164,E2 -22670.164} C_VEL
LIN {X 0,Y 180.088,Z 614.921,A -85,B 0,C 180,E1 -22673.276,E2 -22673.276} C_VEL
LIN {X 0,Y 182.978,Z 613.689,A -85,B 0,C 180,E1 -22676.939,E2 -22676.939} C_VEL
LIN {X 0,Y 186.028,Z 611.715,A -85,B 0,C 180,E1 -22680,E2 -22680} C_VEL
LIN {X 0,Y 190.057,Z 608.502,A -85,B 0,C 180,E1 -22683.28,E2 -22683.28} C_VEL
LIN {X 0,Y 194.449,Z 604.388,A -85,B 0,C 180,E1 -22686.225,E2 -22686.225} C_VEL
LIN {X 0,Y 199.869,Z 598.626,A -85,B 0,C 180,E1 -22689.275,E2 -22689.275} C_VEL
LIN {X 0,Y 205.246,Z 592.12,A -85,B 0,C 180,E1 -22691.856,E2 -22691.856} C_VEL
LIN {X 0,Y 210.888,Z 584.326,A -85,B 0,C 180,E1 -22694.234,E2 -22694.234} C_VEL
LIN {X 0,Y 215.791,Z 576.767,A -85,B 0,C 180,E1 -22696.071,E2 -22696.071} C_VEL
LIN {X 0,Y 221.74,Z 566.275,A -85,B 0,C 180,E1 -22698.049,E2 -22698.049} C_VEL
LIN {X 0,Y 227.096,Z 555.046,A -85,B 0,C 180,E1 -22699.678,E2 -22699.678} C_VEL
LIN {X 0,Y 231.494,Z 544.155,A -85,B 0,C 180,E1 -22700.899,E2 -22700.899} C_VEL
LIN {X 0,Y 235.408,Z 532.242,A -85,B 0,C 180,E1 -22701.926,E2 -22701.926} C_VEL
LIN {X 0,Y 238.845,Z 518.501,A -85,B 0,C 180,E1 -22702.765,E2 -22702.765} C_VEL
LIN {X 0,Y 243.792,Z 489.213,A -85,B 0,C 180,E1 -22703.964,E2 -22703.964} C_VEL
LIN {X 0,Y 244.03,Z 487.272,A -85,B 0,C 180,E1 -22704.1,E2 -22704.1} C_VEL
LIN {X 0,Y 242.398,Z 483.11,A -85,B 0,C 180,E1 -22706.281,E2 -22706.281} C_VEL
LIN {X 0,Y 241.538,Z 481.031,A -85,B 0,C 180,E1 -22707.746,E2 -22707.746} C_VEL
LIN {X 0,Y 240.616,Z 478.639,A -85,B 0,C 180,E1 -22709.951,E2 -22709.951} C_VEL
LIN {X 0,Y 239.872,Z 477.7,A -85,B 0,C 180,E1 -22712.935,E2 -22712.935} C_VEL
LIN {X 0,Y 239.762,Z 477.939,A -85,B 0,C 180,E1 -22713.872,E2 -22713.872} C_VEL
LIN {X 0,Y 239.571,Z 479.484,A -85,B 0,C 180,E1 -22715.24,E2 -22715.24} C_VEL
LIN {X 0,Y 239.388,Z 481.898,A -85,B 0,C 180,E1 -22716.548,E2 -22716.548} C_VEL
LIN {X 0,Y 239.606,Z 487.308,A -85,B 0,C 180,E1 -22719.172,E2 -22719.172} C_VEL
LIN {X 0,Y 239.982,Z 488.671,A -85,B 0,C 180,E1 -22720.082,E2 -22720.082} C_VEL
LIN {X 0,Y 241.277,Z 492.366,A -85,B 0,C 180,E1 -22722.281,E2 -22722.281} C_VEL
LIN {X 0,Y 236.177,Z 521.48,A -85,B 0,C 180,E1 -22723.482,E2 -22723.482} C_VEL
LIN {X 0,Y 232.753,Z 534.581,A -85,B 0,C 180,E1 -22724.186,E2 -22724.186} C_VEL
LIN {X 0,Y 228.103,Z 548.058,A -85,B 0,C 180,E1 -22725.16,E2 -22725.16} C_VEL
LIN {X 0,Y 222.796,Z 560.326,A -85,B 0,C 180,E1 -22726.371,E2 -22726.371} C_VEL
LIN {X 0,Y 217.258,Z 571.078,A -85,B 0,C 180,E1 -22727.841,E2 -22727.841} C_VEL
LIN {X 0,Y 211.348,Z 581.012,A -85,B 0,C 180,E1 -22729.58,E2 -22729.58} C_VEL
LIN {X 0,Y 204.626,Z 590.804,A -85,B 0,C 180,E1 -22731.817,E2 -22731.817} C_VEL
LIN {X 0,Y 197.416,Z 599.927,A -85,B 0,C 180,E1 -22734.658,E2 -22734.658} C_VEL
LIN {X 0,Y 191.741,Z 606.364,A -85,B 0,C 180,E1 -22737.339,E2 -22737.339} C_VEL
LIN {X 0,Y 185.844,Z 612.14,A -85,B 0,C 180,E1 -22740.557,E2 -22740.557} C_VEL
LIN {X 0,Y 180.433,Z 617.124,A -85,B 0,C 180,E1 -22744.634,E2 -22744.634} C_VEL
LIN {X 0,Y 177.969,Z 619.018,A -85,B 0,C 180,E1 -22746.744,E2 -22746.744} C_VEL
LIN {X 0,Y 173.795,Z 621.58,A -85,B 0,C 180,E1 -22751.128,E2 -22751.128} C_VEL
LIN {X 0,Y 171.08,Z 622.66,A -85,B 0,C 180,E1 -22755.734,E2 -22755.734} C_VEL
LIN {X 0,Y 170.154,Z 622.638,A -85,B 0,C 180,E1 -22758.085,E2 -22758.085} C_VEL
LIN {X 0,Y 169.184,Z 621.401,A -85,B 0,C 180,E1 -22762.844,E2 -22762.844} C_VEL
LIN {X 0,Y 169.081,Z 620.423,A -85,B 0,C 180,E1 -22765.085,E2 -22765.085} C_VEL
LIN {X 0,Y 168.947,Z 622.175,A -85,B 0,C 180,E1 -22767.619,E2 -22767.619} C_VEL
LIN {X 0,Y 169.03,Z 623.403,A -85,B 0,C 180,E1 -22770.003,E2 -22770.003} C_VEL
LIN {X 0,Y 168.892,Z 624.298,A -85,B 0,C 180,E1 -22772.924,E2 -22772.924} C_VEL
LIN {X 0,Y 169.094,Z 624.528,A -85,B 0,C 180,E1 -22777.166,E2 -22777.166} C_VEL
LIN {X 0,Y 170.091,Z 623.331,A -85,B 0,C 180,E1 -22781.926,E2 -22781.926} C_VEL
LIN {X 0,Y 170.975,Z 622.121,A -85,B 0,C 180,E1 -22784.281,E2 -22784.281} C_VEL
LIN {X 0,Y 172.796,Z 619.573,A -85,B 0,C 180,E1 -22787.764,E2 -22787.764} C_VEL
LIN {X 0,Y 175.431,Z 616.039,A -85,B 0,C 180,E1 -22791.137,E2 -22791.137} C_VEL
LIN {X 0,Y 178.542,Z 611.451,A -85,B 0,C 180,E1 -22794.416,E2 -22794.416} C_VEL
LIN {X 0,Y 182.119,Z 605.691,A -85,B 0,C 180,E1 -22797.589,E2 -22797.589} C_VEL
LIN {X 0,Y 186.344,Z 598.569,A -85,B 0,C 180,E1 -22800.611,E2 -22800.611} C_VEL
LIN {X 0,Y 191.167,Z 589.78,A -85,B 0,C 180,E1 -22803.47,E2 -22803.47} C_VEL
LIN {X 0,Y 196.099,Z 579.84,A -85,B 0,C 180,E1 -22805.938,E2 -22805.938} C_VEL
LIN {X 0,Y 200.338,Z 569.799,A -85,B 0,C 180,E1 -22807.876,E2 -22807.876} C_VEL
LIN {X 0,Y 204.402,Z 558.775,A -85,B 0,C 180,E1 -22809.504,E2 -22809.504} C_VEL
LIN {X 0,Y 208.075,Z 546.583,A -85,B 0,C 180,E1 -22810.878,E2 -22810.878} C_VEL
LIN {X 0,Y 211.25,Z 533.54,A -85,B 0,C 180,E1 -22811.88,E2 -22811.88} C_VEL
LIN {X 0,Y 213.495,Z 519.629,A -85,B 0,C 180,E1 -22812.646,E2 -22812.646} C_VEL
LIN {X 0,Y 216.93,Z 480.235,A -85,B 0,C 180,E1 -22814.064,E2 -22814.064} C_VEL
LIN {X 0,Y 213.645,Z 471.5,A -85,B 0,C 180,E1 -22815.98,E2 -22815.98} C_VEL
LIN {X 0,Y 210.753,Z 464.905,A -85,B 0,C 180,E1 -22817.778,E2 -22817.778} C_VEL
LIN {X 0,Y 206.825,Z 457.039,A -85,B 0,C 180,E1 -22820.424,E2 -22820.424} C_VEL
LIN {X 0,Y 204.187,Z 452.248,A -85,B 0,C 180,E1 -22822.454,E2 -22822.454} C_VEL
LIN {X 0,Y 201.663,Z 447.804,A -85,B 0,C 180,E1 -22824.625,E2 -22824.625} C_VEL
LIN {X 0,Y 198.861,Z 443.027,A -85,B 0,C 180,E1 -22827.524,E2 -22827.524} C_VEL
LIN {X 0,Y 195.173,Z 437.093,A -85,B 0,C 180,E1 -22832.797,E2 -22832.797} C_VEL
LIN {X 0,Y 193.226,Z 434.645,A -85,B 0,C 180,E1 -22838.111,E2 -22838.111} C_VEL
LIN {X 0,Y 192.939,Z 433.911,A -85,B 0,C 180,E1 -22841.283,E2 -22841.283} C_VEL
LIN {X 0,Y 193.523,Z 434.161,A -85,B 0,C 180,E1 -22845.273,E2 -22845.273} C_VEL
LIN {X 0,Y 195.076,Z 435.401,A -85,B 0,C 180,E1 -22849.097,E2 -22849.097} C_VEL
LIN {X 0,Y 197.142,Z 438.628,A -85,B 0,C 180,E1 -22852.532,E2 -22852.532} C_VEL
LIN {X 0,Y 199.16,Z 440.635,A -85,B 0,C 180,E1 -22854.907,E2 -22854.907} C_VEL
LIN {X 0,Y 202.112,Z 444.745,A -85,B 0,C 180,E1 -22857.836,E2 -22857.836} C_VEL
LIN {X 0,Y 206.098,Z 451.279,A -85,B 0,C 180,E1 -22861.101,E2 -22861.101} C_VEL
LIN {X 0,Y 208.314,Z 455.115,A -85,B 0,C 180,E1 -22862.695,E2 -22862.695} C_VEL
LIN {X 0,Y 212.776,Z 463.616,A -85,B 0,C 180,E1 -22865.542,E2 -22865.542} C_VEL
LIN {X 0,Y 216.961,Z 473.02,A -85,B 0,C 180,E1 -22867.946,E2 -22867.946} C_VEL
LIN {X 0,Y 217.387,Z 474.198,A -85,B 0,C 180,E1 -22868.19,E2 -22868.19} C_VEL
LIN {X 0,Y 213.741,Z 514.32,A -85,B 0,C 180,E1 -22869.627,E2 -22869.627} C_VEL
LIN {X 0,Y 211.673,Z 527.175,A -85,B 0,C 180,E1 -22870.379,E2 -22870.379} C_VEL
LIN {X 0,Y 208.787,Z 539.984,A -85,B 0,C 180,E1 -22871.483,E2 -22871.483} C_VEL
LIN {X 0,Y 205.428,Z 551.42,A -85,B 0,C 180,E1 -22872.822,E2 -22872.822} C_VEL
LIN {X 0,Y 201.369,Z 562.819,A -85,B 0,C 180,E1 -22874.573,E2 -22874.573} C_VEL
LIN {X 0,Y 197.175,Z 572.829,A -85,B 0,C 180,E1 -22876.568,E2 -22876.568} C_VEL
LIN {X 0,Y 192.976,Z 581.455,A -85,B 0,C 180,E1 -22878.75,E2 -22878.75} C_VEL
LIN {X 0,Y 188.637,Z 589.469,A -85,B 0,C 180,E1 -22881.337,E2 -22881.337} C_VEL
LIN {X 0,Y 184.669,Z 596.04,A -85,B 0,C 180,E1 -22884.019,E2 -22884.019} C_VEL
LIN {X 0,Y 181.103,Z 601.436,A -85,B 0,C 180,E1 -22886.799,E2 -22886.799} C_VEL
LIN {X 0,Y 178.008,Z 605.857,A -85,B 0,C 180,E1 -22889.7,E2 -22889.7} C_VEL
LIN {X 0,Y 175.38,Z 609.358,A -85,B 0,C 180,E1 -22892.693,E2 -22892.693} C_VEL
LIN {X 0,Y 173.234,Z 611.996,A -85,B 0,C 180,E1 -22895.764,E2 -22895.764} C_VEL
LIN {X 0,Y 171.492,Z 613.867,A -85,B 0,C 180,E1 -22898.859,E2 -22898.859} C_VEL
LIN {X 0,Y 170.205,Z 615.028,A -85,B 0,C 180,E1 -22901.987,E2 -22901.987} C_VEL
LIN {X 0,Y 169.257,Z 615.443,A -85,B 0,C 180,E1 -22905.095,E2 -22905.095} C_VEL
LIN {X 0,Y 168.623,Z 615.128,A -85,B 0,C 180,E1 -22908.61,E2 -22908.61} C_VEL
LIN {X 0,Y 168.397,Z 613.789,A -85,B 0,C 180,E1 -22912.464,E2 -22912.464} C_VEL
LIN {X 0,Y 168.842,Z 610.658,A -85,B 0,C 180,E1 -22917.237,E2 -22917.237} C_VEL
LIN {X 0,Y 169.82,Z 605.945,A -85,B 0,C 180,E1 -22921.765,E2 -22921.765} C_VEL
LIN {X 0,Y 171.119,Z 600.25,A -85,B 0,C 180,E1 -22925.748,E2 -22925.748} C_VEL
LIN {X 0,Y 172.8,Z 593.632,A -85,B 0,C 180,E1 -22929.3,E2 -22929.3} C_VEL
LIN {X 0,Y 174.701,Z 586.255,A -85,B 0,C 180,E1 -22932.436,E2 -22932.436} C_VEL
LIN {X 0,Y 177.223,Z 576.727,A -85,B 0,C 180,E1 -22935.647,E2 -22935.647} C_VEL
LIN {X 0,Y 179.901,Z 566.159,A -85,B 0,C 180,E1 -22938.427,E2 -22938.427} C_VEL
LIN {X 0,Y 182.496,Z 554.269,A -85,B 0,C 180,E1 -22940.857,E2 -22940.857} C_VEL
LIN {X 0,Y 184.788,Z 542.45,A -85,B 0,C 180,E1 -22942.7,E2 -22942.7} C_VEL
LIN {X 0,Y 186.714,Z 529.609,A -85,B 0,C 180,E1 -22944.191,E2 -22944.191} C_VEL
LIN {X 0,Y 188.172,Z 516.779,A -85,B 0,C 180,E1 -22945.244,E2 -22945.244} C_VEL
LIN {X 0,Y 189.286,Z 501.977,A -85,B 0,C 180,E1 -22945.969,E2 -22945.969} C_VEL
LIN {X 0,Y 191.914,Z 455.409,A -85,B 0,C 180,E1 -22947.803,E2 -22947.803} C_VEL
LIN {X 0,Y 185.213,Z 436.759,A -85,B 0,C 180,E1 -22949.827,E2 -22949.827} C_VEL
LIN {X 0,Y 177.237,Z 420.019,A -85,B 0,C 180,E1 -22952.181,E2 -22952.181} C_VEL
LIN {X 0,Y 173.587,Z 413.778,A -85,B 0,C 180,E1 -22953.264,E2 -22953.264} C_VEL
LIN {X 0,Y 172.116,Z 411.129,A -85,B 0,C 180,E1 -22953.72,E2 -22953.72} C_VEL
LIN {X 0,Y 171.909,Z 410.065,A -85,B 0,C 180,E1 -22953.894,E2 -22953.894} C_VEL
LIN {X 0,Y 171.912,Z 410.072,A -85,B 0,C 180,E1 -22959.408,E2 -22959.408} C_VEL
LIN {X 0,Y 171.61,Z 410.106,A -85,B 0,C 180,E1 -22964.221,E2 -22964.221} C_VEL
LIN {X 0,Y 171.544,Z 410.103,A -85,B 0,C 180,E1 -22969.559,E2 -22969.559} C_VEL
LIN {X 0,Y 171.466,Z 410.116,A -85,B 0,C 180,E1 -22975.613,E2 -22975.613} C_VEL
LIN {X 0,Y 171.436,Z 410.126,A -85,B 0,C 180,E1 -22980.582,E2 -22980.582} C_VEL
LIN {X 0,Y 171.465,Z 410.211,A -85,B 0,C 180,E1 -22983.592,E2 -22983.592} C_VEL
LIN {X 0,Y 180.757,Z 436.402,A -85,B 0,C 180,E1 -22986.167,E2 -22986.167} C_VEL
LIN {X 0,Y 183.946,Z 447.602,A -85,B 0,C 180,E1 -22987.115,E2 -22987.115} C_VEL
LIN {X 0,Y 179.92,Z 512.125,A -85,B 0,C 180,E1 -22990.707,E2 -22990.707} C_VEL
LIN {X 0,Y 178.987,Z 524.341,A -85,B 0,C 180,E1 -22991.751,E2 -22991.751} C_VEL
LIN {X 0,Y 177.569,Z 537.623,A -85,B 0,C 180,E1 -22993.342,E2 -22993.342} C_VEL
LIN {X 0,Y 175.933,Z 550.208,A -85,B 0,C 180,E1 -22995.338,E2 -22995.338} C_VEL
LIN {X 0,Y 174.164,Z 562.449,A -85,B 0,C 180,E1 -22997.866,E2 -22997.866} C_VEL
LIN {X 0,Y 172.756,Z 571.86,A -85,B 0,C 180,E1 -23000.287,E2 -23000.287} C_VEL
LIN {X 0,Y 171.307,Z 581.899,A -85,B 0,C 180,E1 -23003.496,E2 -23003.496} C_VEL
LIN {X 0,Y 170.132,Z 590.665,A -85,B 0,C 180,E1 -23006.986,E2 -23006.986} C_VEL
LIN {X 0,Y 169.372,Z 597.824,A -85,B 0,C 180,E1 -23010.612,E2 -23010.612} C_VEL
LIN {X 0,Y 168.85,Z 603.271,A -85,B 0,C 180,E1 -23014.085,E2 -23014.085} C_VEL
LIN {X 0,Y 168.537,Z 607.982,A -85,B 0,C 180,E1 -23017.957,E2 -23017.957} C_VEL
LIN {X 0,Y 168.58,Z 610.426,A -85,B 0,C 180,E1 -23020.517,E2 -23020.517} C_VEL
LIN {X 0,Y 168.93,Z 612.338,A -85,B 0,C 180,E1 -23023.099,E2 -23023.099} C_VEL
LIN {X 0,Y 169.477,Z 613.75,A -85,B 0,C 180,E1 -23025.592,E2 -23025.592} C_VEL
LIN {X 0,Y 171.159,Z 615.203,A -85,B 0,C 180,E1 -23030.2,E2 -23030.2} C_VEL
LIN {X 0,Y 172.67,Z 615.348,A -85,B 0,C 180,E1 -23032.986,E2 -23032.986} C_VEL
LIN {X 0,Y 175.898,Z 614.494,A -85,B 0,C 180,E1 -23037.209,E2 -23037.209} C_VEL
LIN {X 0,Y 178.591,Z 613.102,A -85,B 0,C 180,E1 -23040,E2 -23040} C_VEL
LIN {X 0,Y 183.11,Z 610.076,A -85,B 0,C 180,E1 -23043.756,E2 -23043.756} C_VEL
LIN {X 0,Y 188.801,Z 605.402,A -85,B 0,C 180,E1 -23047.486,E2 -23047.486} C_VEL
LIN {X 0,Y 195.114,Z 599.18,A -85,B 0,C 180,E1 -23050.9,E2 -23050.9} C_VEL
LIN {X 0,Y 201.226,Z 592.338,A -85,B 0,C 180,E1 -23053.636,E2 -23053.636} C_VEL
LIN {X 0,Y 207.77,Z 583.81,A -85,B 0,C 180,E1 -23056.204,E2 -23056.204} C_VEL
LIN {X 0,Y 213.902,Z 574.687,A -85,B 0,C 180,E1 -23058.287,E2 -23058.287} C_VEL
LIN {X 0,Y 219.865,Z 564.297,A -85,B 0,C 180,E1 -23060.131,E2 -23060.131} C_VEL
LIN {X 0,Y 225.57,Z 552.529,A -85,B 0,C 180,E1 -23061.715,E2 -23061.715} C_VEL
LIN {X 0,Y 231.119,Z 538.319,A -85,B 0,C 180,E1 -23063.124,E2 -23063.124} C_VEL
LIN {X 0,Y 235.188,Z 524.743,A -85,B 0,C 180,E1 -23064.079,E2 -23064.079} C_VEL
LIN {X 0,Y 238.155,Z 511.126,A -85,B 0,C 180,E1 -23064.734,E2 -23064.734} C_VEL
LIN {X 0,Y 241.355,Z 491.932,A -85,B 0,C 180,E1 -23065.493,E2 -23065.493} C_VEL
LIN {X 0,Y 240.061,Z 488.205,A -85,B 0,C 180,E1 -23067.707,E2 -23067.707} C_VEL
LIN {X 0,Y 239.074,Z 485.507,A -85,B 0,C 180,E1 -23070.165,E2 -23070.165} C_VEL
LIN {X 0,Y 238.394,Z 484.633,A -85,B 0,C 180,E1 -23073.176,E2 -23073.176} C_VEL
LIN {X 0,Y 238.558,Z 485.093,A -85,B 0,C 180,E1 -23076.101,E2 -23076.101} C_VEL
LIN {X 0,Y 239.143,Z 486.333,A -85,B 0,C 180,E1 -23078.109,E2 -23078.109} C_VEL
LIN {X 0,Y 239.982,Z 488.671,A -85,B 0,C 180,E1 -23080.082,E2 -23080.082} C_VEL
LIN {X 0,Y 240.078,Z 490.211,A -85,B 0,C 180,E1 -23080.606,E2 -23080.606} C_VEL
LIN {X 0,Y 239.765,Z 493.241,A -85,B 0,C 180,E1 -23080.994,E2 -23080.994} C_VEL
LIN {X 0,Y 239.108,Z 497.056,A -85,B 0,C 180,E1 -23081.168,E2 -23081.168} C_VEL
LIN {X 0,Y 236.938,Z 507.626,A -85,B 0,C 180,E1 -23081.24,E2 -23081.24} C_VEL
LIN {X 0,Y 236.68,Z 509.095,A -85,B 0,C 180,E1 -23081.3,E2 -23081.3} C_VEL
LIN {X 0,Y 233.32,Z 525.555,A -85,B 0,C 180,E1 -23081.988,E2 -23081.988} C_VEL
LIN {X 0,Y 229.075,Z 539.622,A -85,B 0,C 180,E1 -23082.818,E2 -23082.818} C_VEL
LIN {X 0,Y 224.698,Z 550.844,A -85,B 0,C 180,E1 -23083.677,E2 -23083.677} C_VEL
LIN {X 0,Y 218.622,Z 563.462,A -85,B 0,C 180,E1 -23084.994,E2 -23084.994} C_VEL
LIN {X 0,Y 212.307,Z 574.692,A -85,B 0,C 180,E1 -23086.62,E2 -23086.62} C_VEL
LIN {X 0,Y 205.021,Z 585.556,A -85,B 0,C 180,E1 -23088.713,E2 -23088.713} C_VEL
LIN {X 0,Y 198.188,Z 594.386,A -85,B 0,C 180,E1 -23090.995,E2 -23090.995} C_VEL
LIN {X 0,Y 191.803,Z 601.633,A -85,B 0,C 180,E1 -23093.461,E2 -23093.461} C_VEL
LIN {X 0,Y 185.1,Z 608.43,A -85,B 0,C 180,E1 -23096.601,E2 -23096.601} C_VEL
LIN {X 0,Y 179.751,Z 613.092,A -85,B 0,C 180,E1 -23099.454,E2 -23099.454} C_VEL
LIN {X 0,Y 175.404,Z 616.668,A -85,B 0,C 180,E1 -23102.566,E2 -23102.566} C_VEL
LIN {X 0,Y 171.48,Z 619.383,A -85,B 0,C 180,E1 -23105.809,E2 -23105.809} C_VEL
LIN {X 0,Y 167.101,Z 621.679,A -85,B 0,C 180,E1 -23110.342,E2 -23110.342} C_VEL
LIN {X 0,Y 165.415,Z 622.25,A -85,B 0,C 180,E1 -23112.701,E2 -23112.701} C_VEL
LIN {X 0,Y 163.197,Z 622.264,A -85,B 0,C 180,E1 -23117.569,E2 -23117.569} C_VEL
LIN {X 0,Y 162.167,Z 620.825,A -85,B 0,C 180,E1 -23122.533,E2 -23122.533} C_VEL
LIN {X 0,Y 162.051,Z 619.804,A -85,B 0,C 180,E1 -23124.715,E2 -23124.715} C_VEL
LIN {X 0,Y 161.885,Z 621.75,A -85,B 0,C 180,E1 -23127.515,E2 -23127.515} C_VEL
LIN {X 0,Y 161.938,Z 623.027,A -85,B 0,C 180,E1 -23130.003,E2 -23130.003} C_VEL
LIN {X 0,Y 161.797,Z 623.883,A -85,B 0,C 180,E1 -23132.493,E2 -23132.493} C_VEL
LIN {X 0,Y 161.85,Z 624.328,A -85,B 0,C 180,E1 -23134.985,E2 -23134.985} C_VEL
LIN {X 0,Y 162.442,Z 623.994,A -85,B 0,C 180,E1 -23139.969,E2 -23139.969} C_VEL
LIN {X 0,Y 164.081,Z 622.148,A -85,B 0,C 180,E1 -23144.895,E2 -23144.895} C_VEL
LIN {X 0,Y 165.26,Z 620.602,A -85,B 0,C 180,E1 -23147.322,E2 -23147.322} C_VEL
LIN {X 0,Y 167.814,Z 617.518,A -85,B 0,C 180,E1 -23150.856,E2 -23150.856} C_VEL
LIN {X 0,Y 170.94,Z 613.43,A -85,B 0,C 180,E1 -23154.279,E2 -23154.279} C_VEL
LIN {X 0,Y 174.931,Z 607.677,A -85,B 0,C 180,E1 -23157.887,E2 -23157.887} C_VEL
LIN {X 0,Y 179.532,Z 600.556,A -85,B 0,C 180,E1 -23161.247,E2 -23161.247} C_VEL
LIN {X 0,Y 184.417,Z 592.328,A -85,B 0,C 180,E1 -23164.205,E2 -23164.205} C_VEL
LIN {X 0,Y 189.034,Z 583.922,A -85,B 0,C 180,E1 -23166.505,E2 -23166.505} C_VEL
LIN {X 0,Y 193.873,Z 573.701,A -85,B 0,C 180,E1 -23168.709,E2 -23168.709} C_VEL
LIN {X 0,Y 198.531,Z 562.341,A -85,B 0,C 180,E1 -23170.58,E2 -23170.58} C_VEL
LIN {X 0,Y 202.353,Z 551.237,A -85,B 0,C 180,E1 -23171.961,E2 -23171.961} C_VEL
LIN {X 0,Y 205.805,Z 538.784,A -85,B 0,C 180,E1 -23173.08,E2 -23173.08} C_VEL
LIN {X 0,Y 208.598,Z 525.103,A -85,B 0,C 180,E1 -23173.942,E2 -23173.942} C_VEL
LIN {X 0,Y 210.189,Z 511.574,A -85,B 0,C 180,E1 -23174.522,E2 -23174.522} C_VEL
LIN {X 0,Y 212.748,Z 483.011,A -85,B 0,C 180,E1 -23175.522,E2 -23175.522} C_VEL
LIN {X 0,Y 209.82,Z 474.977,A -85,B 0,C 180,E1 -23177.415,E2 -23177.415} C_VEL
LIN {X 0,Y 206.677,Z 467.729,A -85,B 0,C 180,E1 -23179.558,E2 -23179.558} C_VEL
LIN {X 0,Y 203.547,Z 461.367,A -85,B 0,C 180,E1 -23181.935,E2 -23181.935} C_VEL
LIN {X 0,Y 200.09,Z 454.709,A -85,B 0,C 180,E1 -23184.99,E2 -23184.99} C_VEL
LIN {X 0,Y 197.092,Z 449.55,A -85,B 0,C 180,E1 -23188.216,E2 -23188.216} C_VEL
LIN {X 0,Y 193.779,Z 443.831,A -85,B 0,C 180,E1 -23193.43,E2 -23193.43} C_VEL
LIN {X 0,Y 192.076,Z 441.498,A -85,B 0,C 180,E1 -23198.758,E2 -23198.758} C_VEL
LIN {X 0,Y 191.954,Z 440.886,A -85,B 0,C 180,E1 -23202.171,E2 -23202.171} C_VEL
LIN {X 0,Y 192.998,Z 441.576,A -85,B 0,C 180,E1 -23206.845,E2 -23206.845} C_VEL
LIN {X 0,Y 193.822,Z 442.341,A -85,B 0,C 180,E1 -23208.733,E2 -23208.733} C_VEL
LIN {X 0,Y 195.902,Z 445.579,A -85,B 0,C 180,E1 -23212.33,E2 -23212.33} C_VEL
LIN {X 0,Y 197.495,Z 447.279,A -85,B 0,C 180,E1 -23214.331,E2 -23214.331} C_VEL
LIN {X 0,Y 200.228,Z 451.23,A -85,B 0,C 180,E1 -23217.179,E2 -23217.179} C_VEL
LIN {X 0,Y 204.255,Z 458.115,A -85,B 0,C 180,E1 -23220.664,E2 -23220.664} C_VEL
LIN {X 0,Y 207.269,Z 463.948,A -85,B 0,C 180,E1 -23222.916,E2 -23222.916} C_VEL
LIN {X 0,Y 211.04,Z 471.844,A -85,B 0,C 180,E1 -23225.393,E2 -23225.393} C_VEL
LIN {X 0,Y 213.176,Z 476.999,A -85,B 0,C 180,E1 -23226.715,E2 -23226.715} C_VEL
LIN {X 0,Y 209.67,Z 514.13,A -85,B 0,C 180,E1 -23228.046,E2 -23228.046} C_VEL
LIN {X 0,Y 207.468,Z 527.328,A -85,B 0,C 180,E1 -23228.808,E2 -23228.808} C_VEL
LIN {X 0,Y 204.512,Z 540.004,A -85,B 0,C 180,E1 -23229.894,E2 -23229.894} C_VEL
LIN {X 0,Y 200.713,Z 552.297,A -85,B 0,C 180,E1 -23231.344,E2 -23231.344} C_VEL
LIN {X 0,Y 196.419,Z 563.667,A -85,B 0,C 180,E1 -23233.127,E2 -23233.127} C_VEL
LIN {X 0,Y 191.433,Z 574.653,A -85,B 0,C 180,E1 -23235.41,E2 -23235.41} C_VEL
LIN {X 0,Y 186.4,Z 584.297,A -85,B 0,C 180,E1 -23238.03,E2 -23238.03} C_VEL
LIN {X 0,Y 181.806,Z 592.088,A -85,B 0,C 180,E1 -23240.779,E2 -23240.779} C_VEL
LIN {X 0,Y 177.004,Z 599.192,A -85,B 0,C 180,E1 -23244.039,E2 -23244.039} C_VEL
LIN {X 0,Y 173.46,Z 604.049,A -85,B 0,C 180,E1 -23246.949,E2 -23246.949} C_VEL
LIN {X 0,Y 170.366,Z 607.966,A -85,B 0,C 180,E1 -23249.963,E2 -23249.963} C_VEL
LIN {X 0,Y 166.696,Z 612.223,A -85,B 0,C 180,E1 -23254.697,E2 -23254.697} C_VEL
LIN {X 0,Y 164.02,Z 614.759,A -85,B 0,C 180,E1 -23259.527,E2 -23259.527} C_VEL
LIN {X 0,Y 162.501,Z 615.631,A -85,B 0,C 180,E1 -23263.788,E2 -23263.788} C_VEL
LIN {X 0,Y 161.658,Z 615.424,A -85,B 0,C 180,E1 -23267.653,E2 -23267.653} C_VEL
LIN {X 0,Y 161.309,Z 613.845,A -85,B 0,C 180,E1 -23272.41,E2 -23272.41} C_VEL
LIN {X 0,Y 161.745,Z 610.767,A -85,B 0,C 180,E1 -23277.205,E2 -23277.205} C_VEL
LIN {X 0,Y 162.647,Z 606.381,A -85,B 0,C 180,E1 -23281.617,E2 -23281.617} C_VEL
LIN {X 0,Y 164.052,Z 600.427,A -85,B 0,C 180,E1 -23285.981,E2 -23285.981} C_VEL
LIN {X 0,Y 165.777,Z 593.852,A -85,B 0,C 180,E1 -23289.657,E2 -23289.657} C_VEL
LIN {X 0,Y 168.149,Z 585.126,A -85,B 0,C 180,E1 -23293.439,E2 -23293.439} C_VEL
LIN {X 0,Y 170.698,Z 575.805,A -85,B 0,C 180,E1 -23296.606,E2 -23296.606} C_VEL
LIN {X 0,Y 173.214,Z 566.141,A -85,B 0,C 180,E1 -23299.188,E2 -23299.188} C_VEL
LIN {X 0,Y 175.736,Z 555.026,A -85,B 0,C 180,E1 -23301.542,E2 -23301.542} C_VEL
LIN {X 0,Y 178.171,Z 543.099,A -85,B 0,C 180,E1 -23303.485,E2 -23303.485} C_VEL
LIN {X 0,Y 180.067,Z 531.038,A -85,B 0,C 180,E1 -23304.959,E2 -23304.959} C_VEL
LIN {X 0,Y 181.642,Z 517.873,A -85,B 0,C 180,E1 -23306.105,E2 -23306.105} C_VEL
LIN {X 0,Y 182.772,Z 504.407,A -85,B 0,C 180,E1 -23306.823,E2 -23306.823} C_VEL
LIN {X 0,Y 185.517,Z 456.878,A -85,B 0,C 180,E1 -23308.758,E2 -23308.758} C_VEL
LIN {X 0,Y 179.663,Z 440.355,A -85,B 0,C 180,E1 -23310.64,E2 -23310.64} C_VEL
LIN {X 0,Y 171.887,Z 423.885,A -85,B 0,C 180,E1 -23313.045,E2 -23313.045} C_VEL
LIN {X 0,Y 166.276,Z 414.506,A -85,B 0,C 180,E1 -23314.797,E2 -23314.797} C_VEL
LIN {X 0,Y 164.928,Z 411.702,A -85,B 0,C 180,E1 -23315.269,E2 -23315.269} C_VEL
LIN {X 0,Y 164.78,Z 410.96,A -85,B 0,C 180,E1 -23315.35,E2 -23315.35} C_VEL
LIN {X 0,Y 164.854,Z 410.953,A -85,B 0,C 180,E1 -23319.815,E2 -23319.815} C_VEL
LIN {X 0,Y 164.554,Z 410.989,A -85,B 0,C 180,E1 -23324.845,E2 -23324.845} C_VEL
LIN {X 0,Y 164.472,Z 410.984,A -85,B 0,C 180,E1 -23329.986,E2 -23329.986} C_VEL
LIN {X 0,Y 164.391,Z 410.993,A -85,B 0,C 180,E1 -23336.13,E2 -23336.13} C_VEL
LIN {X 0,Y 164.398,Z 411.007,A -85,B 0,C 180,E1 -23342.366,E2 -23342.366} C_VEL
LIN {X 0,Y 164.395,Z 411.007,A -85,B 0,C 180,E1 -23342.799,E2 -23342.799} C_VEL
LIN {X 0,Y 174.188,Z 438.609,A -85,B 0,C 180,E1 -23345.684,E2 -23345.684} C_VEL
LIN {X 0,Y 177.011,Z 448.23,A -85,B 0,C 180,E1 -23346.548,E2 -23346.548} C_VEL
LIN {X 0,Y 172.97,Z 511.991,A -85,B 0,C 180,E1 -23350.251,E2 -23350.251} C_VEL
LIN {X 0,Y 171.863,Z 525.68,A -85,B 0,C 180,E1 -23351.485,E2 -23351.485} C_VEL
LIN {X 0,Y 170.292,Z 540.013,A -85,B 0,C 180,E1 -23353.332,E2 -23353.332} C_VEL
LIN {X 0,Y 168.45,Z 553.42,A -85,B 0,C 180,E1 -23355.681,E2 -23355.681} C_VEL
LIN {X 0,Y 166.708,Z 564.718,A -85,B 0,C 180,E1 -23358.235,E2 -23358.235} C_VEL
LIN {X 0,Y 165.161,Z 574.847,A -85,B 0,C 180,E1 -23361.123,E2 -23361.123} C_VEL
LIN {X 0,Y 163.779,Z 584.668,A -85,B 0,C 180,E1 -23364.613,E2 -23364.613} C_VEL
LIN {X 0,Y 162.76,Z 592.435,A -85,B 0,C 180,E1 -23368.065,E2 -23368.065} C_VEL
LIN {X 0,Y 162.166,Z 598.761,A -85,B 0,C 180,E1 -23371.528,E2 -23371.528} C_VEL
LIN {X 0,Y 161.648,Z 604.183,A -85,B 0,C 180,E1 -23375.245,E2 -23375.245} C_VEL
LIN {X 0,Y 161.486,Z 609.052,A -85,B 0,C 180,E1 -23379.624,E2 -23379.624} C_VEL
LIN {X 0,Y 161.795,Z 611.685,A -85,B 0,C 180,E1 -23382.856,E2 -23382.856} C_VEL
LIN {X 0,Y 162.923,Z 614.308,A -85,B 0,C 180,E1 -23387.544,E2 -23387.544} C_VEL
LIN {X 0,Y 164.01,Z 615.161,A -85,B 0,C 180,E1 -23390.234,E2 -23390.234} C_VEL
LIN {X 0,Y 166.892,Z 615.565,A -85,B 0,C 180,E1 -23395.168,E2 -23395.168} C_VEL
LIN {X 0,Y 168.896,Z 615.112,A -85,B 0,C 180,E1 -23397.615,E2 -23397.615} C_VEL
LIN {X 0,Y 171.132,Z 614.254,A -85,B 0,C 180,E1 -23400,E2 -23400} C_VEL
LIN {X 0,Y 176.177,Z 611.545,A -85,B 0,C 180,E1 -23404.266,E2 -23404.266} C_VEL
LIN {X 0,Y 181.464,Z 607.813,A -85,B 0,C 180,E1 -23407.79,E2 -23407.79} C_VEL
LIN {X 0,Y 186.941,Z 603.226,A -85,B 0,C 180,E1 -23410.834,E2 -23410.834} C_VEL
LIN {X 0,Y 193.021,Z 597.368,A -85,B 0,C 180,E1 -23413.69,E2 -23413.69} C_VEL
LIN {X 0,Y 199.703,Z 589.996,A -85,B 0,C 180,E1 -23416.352,E2 -23416.352} C_VEL
LIN {X 0,Y 205.684,Z 582.435,A -85,B 0,C 180,E1 -23418.476,E2 -23418.476} C_VEL
LIN {X 0,Y 212.052,Z 573.153,A -85,B 0,C 180,E1 -23420.447,E2 -23420.447} C_VEL
LIN {X 0,Y 218.344,Z 562.458,A -85,B 0,C 180,E1 -23422.222,E2 -23422.222} C_VEL
LIN {X 0,Y 224.148,Z 550.642,A -85,B 0,C 180,E1 -23423.697,E2 -23423.697} C_VEL
LIN {X 0,Y 228.656,Z 539.451,A -85,B 0,C 180,E1 -23424.757,E2 -23424.757} C_VEL
LIN {X 0,Y 232.534,Z 527.515,A -85,B 0,C 180,E1 -23425.593,E2 -23425.593} C_VEL
LIN {X 0,Y 235.51,Z 515.438,A -85,B 0,C 180,E1 -23426.225,E2 -23426.225} C_VEL
LIN {X 0,Y 238.918,Z 496.614,A -85,B 0,C 180,E1 -23426.976,E2 -23426.976} C_VEL
LIN {X 0,Y 238.051,Z 494.129,A -85,B 0,C 180,E1 -23428.759,E2 -23428.759} C_VEL
LIN {X 0,Y 237.456,Z 492.312,A -85,B 0,C 180,E1 -23430.575,E2 -23430.575} C_VEL
LIN {X 0,Y 236.926,Z 491.547,A -85,B 0,C 180,E1 -23433.847,E2 -23433.847} C_VEL
LIN {X 0,Y 237.167,Z 492.184,A -85,B 0,C 180,E1 -23436.346,E2 -23436.346} C_VEL
LIN {X 0,Y 237.56,Z 493.148,A -85,B 0,C 180,E1 -23437.777,E2 -23437.777} C_VEL
LIN {X 0,Y 238.486,Z 496.149,A -85,B 0,C 180,E1 -23440.181,E2 -23440.181} C_VEL
LIN {X 0,Y 238.777,Z 497.23,A -85,B 0,C 180,E1 -23440.822,E2 -23440.822} C_VEL
LIN {X 0,Y 236.68,Z 509.095,A -85,B 0,C 180,E1 -23441.3,E2 -23441.3} C_VEL
LIN {X 0,Y 235.52,Z 514.878,A -85,B 0,C 180,E1 -23441.385,E2 -23441.385} C_VEL
LIN {X 0,Y 232.759,Z 524.316,A -85,B 0,C 180,E1 -23441.044,E2 -23441.044} C_VEL
LIN {X 0,Y 229.462,Z 533.676,A -85,B 0,C 180,E1 -23440.838,E2 -23440.838} C_VEL
LIN {X 0,Y 227.471,Z 539.11,A -85,B 0,C 180,E1 -23441.037,E2 -23441.037} C_VEL
LIN {X 0,Y 222.465,Z 551.372,A -85,B 0,C 180,E1 -23441.95,E2 -23441.95} C_VEL
LIN {X 0,Y 216.081,Z 564.086,A -85,B 0,C 180,E1 -23443.239,E2 -23443.239} C_VEL
LIN {X 0,Y 210.029,Z 574.234,A -85,B 0,C 180,E1 -23444.682,E2 -23444.682} C_VEL
LIN {X 0,Y 202.403,Z 585.08,A -85,B 0,C 180,E1 -23446.707,E2 -23446.707} C_VEL
LIN {X 0,Y 195.19,Z 593.939,A -85,B 0,C 180,E1 -23448.924,E2 -23448.924} C_VEL
LIN {X 0,Y 187.334,Z 602.235,A -85,B 0,C 180,E1 -23451.76,E2 -23451.76} C_VEL
LIN {X 0,Y 181.228,Z 607.994,A -85,B 0,C 180,E1 -23454.434,E2 -23454.434} C_VEL
LIN {X 0,Y 175.569,Z 612.632,A -85,B 0,C 180,E1 -23457.293,E2 -23457.293} C_VEL
LIN {X 0,Y 172.173,Z 615.189,A -85,B 0,C 180,E1 -23459.324,E2 -23459.324} C_VEL
LIN {X 0,Y 167.744,Z 618.203,A -85,B 0,C 180,E1 -23462.561,E2 -23462.561} C_VEL
LIN {X 0,Y 162.566,Z 620.904,A -85,B 0,C 180,E1 -23467.106,E2 -23467.106} C_VEL
LIN {X 0,Y 158.63,Z 622.112,A -85,B 0,C 180,E1 -23471.936,E2 -23471.936} C_VEL
LIN {X 0,Y 156.262,Z 621.888,A -85,B 0,C 180,E1 -23477.008,E2 -23477.008} C_VEL
LIN {X 0,Y 155.163,Z 620.126,A -85,B 0,C 180,E1 -23482.194,E2 -23482.194} C_VEL
LIN {X 0,Y 155.013,Z 619.123,A -85,B 0,C 180,E1 -23484.312,E2 -23484.312} C_VEL
LIN {X 0,Y 154.815,Z 621.308,A -85,B 0,C 180,E1 -23487.402,E2 -23487.402} C_VEL
LIN {X 0,Y 154.873,Z 622.637,A -85,B 0,C 180,E1 -23490.003,E2 -23490.003} C_VEL
LIN {X 0,Y 154.716,Z 623.543,A -85,B 0,C 180,E1 -23492.607,E2 -23492.607} C_VEL
LIN {X 0,Y 154.759,Z 624.06,A -85,B 0,C 180,E1 -23495.214,E2 -23495.214} C_VEL
LIN {X 0,Y 154.97,Z 624.172,A -85,B 0,C 180,E1 -23497.823,E2 -23497.823} C_VEL
LIN {X 0,Y 156.188,Z 623.192,A -85,B 0,C 180,E1 -23503.005,E2 -23503.005} C_VEL
LIN {X 0,Y 158.478,Z 620.699,A -85,B 0,C 180,E1 -23508.088,E2 -23508.088} C_VEL
LIN {X 0,Y 161.199,Z 617.729,A -85,B 0,C 180,E1 -23511.755,E2 -23511.755} C_VEL
LIN {X 0,Y 164.485,Z 613.766,A -85,B 0,C 180,E1 -23515.298,E2 -23515.298} C_VEL
LIN {X 0,Y 168.586,Z 608.385,A -85,B 0,C 180,E1 -23518.902,E2 -23518.902} C_VEL
LIN {X 0,Y 173.551,Z 601.241,A -85,B 0,C 180,E1 -23522.453,E2 -23522.453} C_VEL
LIN {X 0,Y 178.643,Z 593.243,A -85,B 0,C 180,E1 -23525.473,E2 -23525.473} C_VEL
LIN {X 0,Y 183.445,Z 585.114,A -85,B 0,C 180,E1 -23527.809,E2 -23527.809} C_VEL
LIN {X 0,Y 188.466,Z 575.305,A -85,B 0,C 180,E1 -23530.039,E2 -23530.039} C_VEL
LIN {X 0,Y 193.304,Z 564.327,A -85,B 0,C 180,E1 -23531.921,E2 -23531.921} C_VEL
LIN {X 0,Y 197.817,Z 552.039,A -85,B 0,C 180,E1 -23533.503,E2 -23533.503} C_VEL
LIN {X 0,Y 201.234,Z 540.51,A -85,B 0,C 180,E1 -23534.588,E2 -23534.588} C_VEL
LIN {X 0,Y 204.287,Z 526.8,A -85,B 0,C 180,E1 -23535.475,E2 -23535.475} C_VEL
LIN {X 0,Y 206.105,Z 513.642,A -85,B 0,C 180,E1 -23536.077,E2 -23536.077} C_VEL
LIN {X 0,Y 208.725,Z 485.821,A -85,B 0,C 180,E1 -23537.062,E2 -23537.062} C_VEL
LIN {X 0,Y 206.08,Z 478.325,A -85,B 0,C 180,E1 -23538.957,E2 -23538.957} C_VEL
LIN {X 0,Y 202.965,Z 471.148,A -85,B 0,C 180,E1 -23541.325,E2 -23541.325} C_VEL
LIN {X 0,Y 199.975,Z 464.854,A -85,B 0,C 180,E1 -23543.887,E2 -23543.887} C_VEL
LIN {X 0,Y 197.677,Z 460.301,A -85,B 0,C 180,E1 -23546.216,E2 -23546.216} C_VEL
LIN {X 0,Y 195.416,Z 456.036,A -85,B 0,C 180,E1 -23548.911,E2 -23548.911} C_VEL
LIN {X 0,Y 192.55,Z 450.733,A -85,B 0,C 180,E1 -23553.765,E2 -23553.765} C_VEL
LIN {X 0,Y 191.041,Z 448.577,A -85,B 0,C 180,E1 -23558.638,E2 -23558.638} C_VEL
LIN {X 0,Y 190.869,Z 448.03,A -85,B 0,C 180,E1 -23560.647,E2 -23560.647} C_VEL
LIN {X 0,Y 191.157,Z 447.994,A -85,B 0,C 180,E1 -23563.992,E2 -23563.992} C_VEL
LIN {X 0,Y 192.523,Z 449.102,A -85,B 0,C 180,E1 -23568.211,E2 -23568.211} C_VEL
LIN {X 0,Y 194.476,Z 452.377,A -85,B 0,C 180,E1 -23571.872,E2 -23571.872} C_VEL
LIN {X 0,Y 195.958,Z 454.032,A -85,B 0,C 180,E1 -23573.824,E2 -23573.824} C_VEL
LIN {X 0,Y 198.358,Z 457.699,A -85,B 0,C 180,E1 -23576.499,E2 -23576.499} C_VEL
LIN {X 0,Y 202.438,Z 464.979,A -85,B 0,C 180,E1 -23580.231,E2 -23580.231} C_VEL
LIN {X 0,Y 206.583,Z 473.822,A -85,B 0,C 180,E1 -23583.409,E2 -23583.409} C_VEL
LIN {X 0,Y 209.12,Z 479.923,A -85,B 0,C 180,E1 -23585.143,E2 -23585.143} C_VEL
LIN {X 0,Y 205.637,Z 515.11,A -85,B 0,C 180,E1 -23586.453,E2 -23586.453} C_VEL
LIN {X 0,Y 203.339,Z 528.026,A -85,B 0,C 180,E1 -23587.209,E2 -23587.209} C_VEL
LIN {X 0,Y 200.338,Z 540.238,A -85,B 0,C 180,E1 -23588.262,E2 -23588.262} C_VEL
LIN {X 0,Y 196.56,Z 552.076,A -85,B 0,C 180,E1 -23589.651,E2 -23589.651} C_VEL
LIN {X 0,Y 191.948,Z 563.822,A -85,B 0,C 180,E1 -23591.48,E2 -23591.48} C_VEL
LIN {X 0,Y 187.099,Z 574.11,A -85,B 0,C 180,E1 -23593.596,E2 -23593.596} C_VEL
LIN {X 0,Y 181.965,Z 583.472,A -85,B 0,C 180,E1 -23596.099,E2 -23596.099} C_VEL
LIN {X 0,Y 176.62,Z 592.073,A -85,B 0,C 180,E1 -23599.112,E2 -23599.112} C_VEL
LIN {X 0,Y 171.089,Z 599.78,A -85,B 0,C 180,E1 -23602.74,E2 -23602.74} C_VEL
LIN {X 0,Y 167.19,Z 604.756,A -85,B 0,C 180,E1 -23605.865,E2 -23605.865} C_VEL
LIN {X 0,Y 162.751,Z 609.871,A -85,B 0,C 180,E1 -23610.266,E2 -23610.266} C_VEL
LIN {X 0,Y 159.26,Z 613.378,A -85,B 0,C 180,E1 -23615.007,E2 -23615.007} C_VEL
LIN {X 0,Y 156.564,Z 615.467,A -85,B 0,C 180,E1 -23620.256,E2 -23620.256} C_VEL
LIN {X 0,Y 155.412,Z 615.872,A -85,B 0,C 180,E1 -23623.647,E2 -23623.647} C_VEL
LIN {X 0,Y 154.664,Z 615.633,A -85,B 0,C 180,E1 -23627.027,E2 -23627.027} C_VEL
LIN {X 0,Y 154.236,Z 614.597,A -85,B 0,C 180,E1 -23630.772,E2 -23630.772} C_VEL
LIN {X 0,Y 154.327,Z 612.366,A -85,B 0,C 180,E1 -23635.057,E2 -23635.057} C_VEL
LIN {X 0,Y 155.028,Z 608.822,A -85,B 0,C 180,E1 -23639.468,E2 -23639.468} C_VEL
LIN {X 0,Y 155.947,Z 604.729,A -85,B 0,C 180,E1 -23643.21,E2 -23643.21} C_VEL
LIN {X 0,Y 157.605,Z 598.267,A -85,B 0,C 180,E1 -23647.677,E2 -23647.677} C_VEL
LIN {X 0,Y 159.552,Z 591.351,A -85,B 0,C 180,E1 -23651.373,E2 -23651.373} C_VEL
LIN {X 0,Y 161.913,Z 582.941,A -85,B 0,C 180,E1 -23654.901,E2 -23654.901} C_VEL
LIN {X 0,Y 164.697,Z 573.09,A -85,B 0,C 180,E1 -23658.141,E2 -23658.141} C_VEL
LIN {X 0,Y 167.153,Z 563.596,A -85,B 0,C 180,E1 -23660.62,E2 -23660.62} C_VEL
LIN {X 0,Y 169.699,Z 552.732,A -85,B 0,C 180,E1 -23662.86,E2 -23662.86} C_VEL
LIN {X 0,Y 172.229,Z 539.87,A -85,B 0,C 180,E1 -23664.876,E2 -23664.876} C_VEL
LIN {X 0,Y 174.22,Z 526.997,A -85,B 0,C 180,E1 -23666.351,E2 -23666.351} C_VEL
LIN {X 0,Y 175.715,Z 513.653,A -85,B 0,C 180,E1 -23667.38,E2 -23667.38} C_VEL
LIN {X 0,Y 177.59,Z 485.178,A -85,B 0,C 180,E1 -23668.653,E2 -23668.653} C_VEL
LIN {X 0,Y 179.151,Z 458.374,A -85,B 0,C 180,E1 -23669.785,E2 -23669.785} C_VEL
LIN {X 0,Y 173.978,Z 443.717,A -85,B 0,C 180,E1 -23671.525,E2 -23671.525} C_VEL
LIN {X 0,Y 166.673,Z 427.974,A -85,B 0,C 180,E1 -23673.919,E2 -23673.919} C_VEL
LIN {X 0,Y 159.862,Z 416.198,A -85,B 0,C 180,E1 -23676.197,E2 -23676.197} C_VEL
LIN {X 0,Y 158.126,Z 413.222,A -85,B 0,C 180,E1 -23676.817,E2 -23676.817} C_VEL
LIN {X 0,Y 157.801,Z 411.821,A -85,B 0,C 180,E1 -23677.032,E2 -23677.032} C_VEL
LIN {X 0,Y 157.706,Z 411.836,A -85,B 0,C 180,E1 -23681.359,E2 -23681.359} C_VEL
LIN {X 0,Y 157.479,Z 411.871,A -85,B 0,C 180,E1 -23685.528,E2 -23685.528} C_VEL
LIN {X 0,Y 157.369,Z 411.875,A -85,B 0,C 180,E1 -23690.929,E2 -23690.929} C_VEL
LIN {X 0,Y 157.311,Z 411.87,A -85,B 0,C 180,E1 -23696.68,E2 -23696.68} C_VEL
LIN {X 0,Y 157.394,Z 412.031,A -85,B 0,C 180,E1 -23702.079,E2 -23702.079} C_VEL
LIN {X 0,Y 167.682,Z 440.984,A -85,B 0,C 180,E1 -23705.186,E2 -23705.186} C_VEL
LIN {X 0,Y 170.097,Z 449.372,A -85,B 0,C 180,E1 -23705.978,E2 -23705.978} C_VEL
LIN {X 0,Y 166.034,Z 511.994,A -85,B 0,C 180,E1 -23709.773,E2 -23709.773} C_VEL
LIN {X 0,Y 164.869,Z 525.722,A -85,B 0,C 180,E1 -23711.063,E2 -23711.063} C_VEL
LIN {X 0,Y 163.271,Z 539.86,A -85,B 0,C 180,E1 -23712.965,E2 -23712.965} C_VEL
LIN {X 0,Y 161.602,Z 551.767,A -85,B 0,C 180,E1 -23715.105,E2 -23715.105} C_VEL
LIN {X 0,Y 159.937,Z 562.495,A -85,B 0,C 180,E1 -23717.541,E2 -23717.541} C_VEL
LIN {X 0,Y 158.385,Z 572.536,A -85,B 0,C 180,E1 -23720.367,E2 -23720.367} C_VEL
LIN {X 0,Y 157.059,Z 581.91,A -85,B 0,C 180,E1 -23723.648,E2 -23723.648} C_VEL
LIN {X 0,Y 155.916,Z 590.27,A -85,B 0,C 180,E1 -23727.254,E2 -23727.254} C_VEL
LIN {X 0,Y 155.193,Z 597.047,A -85,B 0,C 180,E1 -23730.868,E2 -23730.868} C_VEL
LIN {X 0,Y 154.692,Z 602.312,A -85,B 0,C 180,E1 -23734.361,E2 -23734.361} C_VEL
LIN {X 0,Y 154.385,Z 607.372,A -85,B 0,C 180,E1 -23738.643,E2 -23738.643} C_VEL
LIN {X 0,Y 154.664,Z 610.901,A -85,B 0,C 180,E1 -23742.588,E2 -23742.588} C_VEL
LIN {X 0,Y 155.61,Z 613.657,A -85,B 0,C 180,E1 -23746.949,E2 -23746.949} C_VEL
LIN {X 0,Y 157.837,Z 615.527,A -85,B 0,C 180,E1 -23752.323,E2 -23752.323} C_VEL
LIN {X 0,Y 159.428,Z 615.85,A -85,B 0,C 180,E1 -23754.942,E2 -23754.942} C_VEL
LIN {X 0,Y 163.693,Z 615.181,A -85,B 0,C 180,E1 -23760,E2 -23760} C_VEL
LIN {X 0,Y 166.294,Z 614.25,A -85,B 0,C 180,E1 -23762.422,E2 -23762.422} C_VEL
LIN {X 0,Y 169.263,Z 612.822,A -85,B 0,C 180,E1 -23764.831,E2 -23764.831} C_VEL
LIN {X 0,Y 174.102,Z 609.975,A -85,B 0,C 180,E1 -23768.122,E2 -23768.122} C_VEL
LIN {X 0,Y 179.709,Z 605.998,A -85,B 0,C 180,E1 -23771.276,E2 -23771.276} C_VEL
LIN {X 0,Y 186.992,Z 599.822,A -85,B 0,C 180,E1 -23774.696,E2 -23774.696} C_VEL
LIN {X 0,Y 193.845,Z 593.088,A -85,B 0,C 180,E1 -23777.404,E2 -23777.404} C_VEL
LIN {X 0,Y 201.327,Z 584.429,A -85,B 0,C 180,E1 -23779.952,E2 -23779.952} C_VEL
LIN {X 0,Y 207.786,Z 575.924,A -85,B 0,C 180,E1 -23781.842,E2 -23781.842} C_VEL
LIN {X 0,Y 214.1,Z 566.144,A -85,B 0,C 180,E1 -23783.551,E2 -23783.551} C_VEL
LIN {X 0,Y 220.849,Z 553.636,A -85,B 0,C 180,E1 -23785.19,E2 -23785.19} C_VEL
LIN {X 0,Y 226.477,Z 540.756,A -85,B 0,C 180,E1 -23786.425,E2 -23786.425} C_VEL
LIN {X 0,Y 231.019,Z 527.435,A -85,B 0,C 180,E1 -23787.343,E2 -23787.343} C_VEL
LIN {X 0,Y 234.234,Z 514.571,A -85,B 0,C 180,E1 -23787.961,E2 -23787.961} C_VEL
LIN {X 0,Y 236.658,Z 501.618,A -85,B 0,C 180,E1 -23788.478,E2 -23788.478} C_VEL
LIN {X 0,Y 235.926,Z 499.169,A -85,B 0,C 180,E1 -23790.795,E2 -23790.795} C_VEL
LIN {X 0,Y 235.483,Z 498.537,A -85,B 0,C 180,E1 -23793.32,E2 -23793.32} C_VEL
LIN {X 0,Y 235.636,Z 498.982,A -85,B 0,C 180,E1 -23795.978,E2 -23795.978} C_VEL
LIN {X 0,Y 235.963,Z 499.812,A -85,B 0,C 180,E1 -23797.321,E2 -23797.321} C_VEL
LIN {X 0,Y 236.569,Z 502.05,A -85,B 0,C 180,E1 -23799.287,E2 -23799.287} C_VEL
LIN {X 0,Y 232.678,Z 521.926,A -85,B 0,C 180,E1 -23800.117,E2 -23800.117} C_VEL
LIN {X 0,Y 229.404,Z 533.454,A -85,B 0,C 180,E1 -23800.683,E2 -23800.683} C_VEL
LIN {X 0,Y 227.471,Z 539.11,A -85,B 0,C 180,E1 -23801.037,E2 -23801.037} C_VEL
LIN {X 0,Y 225.268,Z 544.533,A -85,B 0,C 180,E1 -23801.26,E2 -23801.26} C_VEL
LIN {X 0,Y 220.701,Z 553.362,A -85,B 0,C 180,E1 -23801.232,E2 -23801.232} C_VEL
LIN {X 0,Y 215.631,Z 561.853,A -85,B 0,C 180,E1 -23801.297,E2 -23801.297} C_VEL
LIN {X 0,Y 212.645,Z 566.655,A -85,B 0,C 180,E1 -23801.68,E2 -23801.68} C_VEL
LIN {X 0,Y 205.343,Z 577.823,A -85,B 0,C 180,E1 -23803.344,E2 -23803.344} C_VEL
LIN {X 0,Y 197.636,Z 587.736,A -85,B 0,C 180,E1 -23805.319,E2 -23805.319} C_VEL
LIN {X 0,Y 190.072,Z 596.128,A -85,B 0,C 180,E1 -23807.565,E2 -23807.565} C_VEL
LIN {X 0,Y 183.059,Z 602.952,A -85,B 0,C 180,E1 -23809.983,E2 -23809.983} C_VEL
LIN {X 0,Y 175.6,Z 609.258,A -85,B 0,C 180,E1 -23813.11,E2 -23813.11} C_VEL
LIN {X 0,Y 167.787,Z 614.843,A -85,B 0,C 180,E1 -23817.012,E2 -23817.012} C_VEL
LIN {X 0,Y 161.48,Z 618.661,A -85,B 0,C 180,E1 -23821.4,E2 -23821.4} C_VEL
LIN {X 0,Y 156.067,Z 621.036,A -85,B 0,C 180,E1 -23826.095,E2 -23826.095} C_VEL
LIN {X 0,Y 151.879,Z 621.955,A -85,B 0,C 180,E1 -23831.104,E2 -23831.104} C_VEL
LIN {X 0,Y 149.35,Z 621.392,A -85,B 0,C 180,E1 -23836.395,E2 -23836.395} C_VEL
LIN {X 0,Y 148.154,Z 619.4,A -85,B 0,C 180,E1 -23841.822,E2 -23841.822} C_VEL
LIN {X 0,Y 147.982,Z 618.423,A -85,B 0,C 180,E1 -23843.869,E2 -23843.869} C_VEL
LIN {X 0,Y 147.721,Z 621.008,A -85,B 0,C 180,E1 -23847.567,E2 -23847.567} C_VEL
LIN {X 0,Y 147.779,Z 622.242,A -85,B 0,C 180,E1 -23850.004,E2 -23850.004} C_VEL
LIN {X 0,Y 147.638,Z 623.203,A -85,B 0,C 180,E1 -23852.732,E2 -23852.732} C_VEL
LIN {X 0,Y 147.69,Z 623.774,A -85,B 0,C 180,E1 -23855.465,E2 -23855.465} C_VEL
LIN {X 0,Y 147.939,Z 623.961,A -85,B 0,C 180,E1 -23858.197,E2 -23858.197} C_VEL
LIN {X 0,Y 148.432,Z 623.75,A -85,B 0,C 180,E1 -23860.921,E2 -23860.921} C_VEL
LIN {X 0,Y 150.321,Z 622.14,A -85,B 0,C 180,E1 -23866.295,E2 -23866.295} C_VEL
LIN {X 0,Y 151.733,Z 620.768,A -85,B 0,C 180,E1 -23868.922,E2 -23868.922} C_VEL
LIN {X 0,Y 154.633,Z 617.917,A -85,B 0,C 180,E1 -23872.729,E2 -23872.729} C_VEL
LIN {X 0,Y 158.085,Z 614.086,A -85,B 0,C 180,E1 -23876.399,E2 -23876.399} C_VEL
LIN {X 0,Y 162.126,Z 609.225,A -85,B 0,C 180,E1 -23879.891,E2 -23879.891} C_VEL
LIN {X 0,Y 166.817,Z 603.129,A -85,B 0,C 180,E1 -23883.212,E2 -23883.212} C_VEL
LIN {X 0,Y 172.084,Z 595.635,A -85,B 0,C 180,E1 -23886.316,E2 -23886.316} C_VEL
LIN {X 0,Y 177.955,Z 586.312,A -85,B 0,C 180,E1 -23889.193,E2 -23889.193} C_VEL
LIN {X 0,Y 183.712,Z 575.725,A -85,B 0,C 180,E1 -23891.662,E2 -23891.662} C_VEL
LIN {X 0,Y 188.75,Z 565.006,A -85,B 0,C 180,E1 -23893.541,E2 -23893.541} C_VEL
LIN {X 0,Y 193.43,Z 552.996,A -85,B 0,C 180,E1 -23895.117,E2 -23895.117} C_VEL
LIN {X 0,Y 197.338,Z 540.647,A -85,B 0,C 180,E1 -23896.287,E2 -23896.287} C_VEL
LIN {X 0,Y 200.455,Z 527.305,A -85,B 0,C 180,E1 -23897.161,E2 -23897.161} C_VEL
LIN {X 0,Y 202.43,Z 513.817,A -85,B 0,C 180,E1 -23897.782,E2 -23897.782} C_VEL
LIN {X 0,Y 204.871,Z 488.472,A -85,B 0,C 180,E1 -23898.705,E2 -23898.705} C_VEL
LIN {X 0,Y 202.338,Z 481.381,A -85,B 0,C 180,E1 -23900.705,E2 -23900.705} C_VEL
LIN {X 0,Y 199.165,Z 473.835,A -85,B 0,C 180,E1 -23903.46,E2 -23903.46} C_VEL
LIN {X 0,Y 196.173,Z 467.253,A -85,B 0,C 180,E1 -23906.567,E2 -23906.567} C_VEL
LIN {X 0,Y 193.774,Z 462.577,A -85,B 0,C 180,E1 -23909.611,E2 -23909.611} C_VEL
LIN {X 0,Y 191.301,Z 457.602,A -85,B 0,C 180,E1 -23914.166,E2 -23914.166} C_VEL
LIN {X 0,Y 189.939,Z 455.505,A -85,B 0,C 180,E1 -23919.036,E2 -23919.036} C_VEL
LIN {X 0,Y 189.926,Z 454.937,A -85,B 0,C 180,E1 -23922.781,E2 -23922.781} C_VEL
LIN {X 0,Y 191.048,Z 455.774,A -85,B 0,C 180,E1 -23927.249,E2 -23927.249} C_VEL
LIN {X 0,Y 191.611,Z 456.835,A -85,B 0,C 180,E1 -23928.687,E2 -23928.687} C_VEL
LIN {X 0,Y 193.661,Z 459.76,A -85,B 0,C 180,E1 -23932.248,E2 -23932.248} C_VEL
LIN {X 0,Y 194.551,Z 460.959,A -85,B 0,C 180,E1 -23933.461,E2 -23933.461} C_VEL
LIN {X 0,Y 196.602,Z 464.31,A -85,B 0,C 180,E1 -23935.9,E2 -23935.9} C_VEL
LIN {X 0,Y 200.186,Z 471.105,A -85,B 0,C 180,E1 -23939.425,E2 -23939.425} C_VEL
LIN {X 0,Y 204.03,Z 479.828,A -85,B 0,C 180,E1 -23942.603,E2 -23942.603} C_VEL
LIN {X 0,Y 205.35,Z 483.178,A -85,B 0,C 180,E1 -23943.581,E2 -23943.581} C_VEL
LIN {X 0,Y 202.001,Z 515.081,A -85,B 0,C 180,E1 -23944.738,E2 -23944.738} C_VEL
LIN {X 0,Y 199.626,Z 528.014,A -85,B 0,C 180,E1 -23945.48,E2 -23945.48} C_VEL
LIN {X 0,Y 196.328,Z 540.858,A -85,B 0,C 180,E1 -23946.582,E2 -23946.582} C_VEL
LIN {X 0,Y 192.482,Z 552.317,A -85,B 0,C 180,E1 -23947.929,E2 -23947.929} C_VEL
LIN {X 0,Y 188.009,Z 563.206,A -85,B 0,C 180,E1 -23949.61,E2 -23949.61} C_VEL
LIN {X 0,Y 183.004,Z 573.461,A -85,B 0,C 180,E1 -23951.669,E2 -23951.669} C_VEL
LIN {X 0,Y 177.524,Z 583.025,A -85,B 0,C 180,E1 -23954.173,E2 -23954.173} C_VEL
LIN {X 0,Y 172.346,Z 591.054,A -85,B 0,C 180,E1 -23956.94,E2 -23956.94} C_VEL
LIN {X 0,Y 166.838,Z 598.534,A -85,B 0,C 180,E1 -23960.306,E2 -23960.306} C_VEL
LIN {X 0,Y 161.68,Z 604.679,A -85,B 0,C 180,E1 -23964.092,E2 -23964.092} C_VEL
LIN {X 0,Y 156.85,Z 609.844,A -85,B 0,C 180,E1 -23968.594,E2 -23968.594} C_VEL
LIN {X 0,Y 152.989,Z 613.441,A -85,B 0,C 180,E1 -23973.454,E2 -23973.454} C_VEL
LIN {X 0,Y 150.627,Z 615.219,A -85,B 0,C 180,E1 -23977.51,E2 -23977.51} C_VEL
LIN {X 0,Y 148.988,Z 616.022,A -85,B 0,C 180,E1 -23981.331,E2 -23981.331} C_VEL
LIN {X 0,Y 147.806,Z 615.968,A -85,B 0,C 180,E1 -23985.499,E2 -23985.499} C_VEL
LIN {X 0,Y 147.195,Z 614.952,A -85,B 0,C 180,E1 -23989.813,E2 -23989.813} C_VEL
LIN {X 0,Y 147.242,Z 612.364,A -85,B 0,C 180,E1 -23995.052,E2 -23995.052} C_VEL
LIN {X 0,Y 147.796,Z 609.496,A -85,B 0,C 180,E1 -23998.864,E2 -23998.864} C_VEL
LIN {X 0,Y 148.972,Z 604.443,A -85,B 0,C 180,E1 -24003.685,E2 -24003.685} C_VEL
LIN {X 0,Y 150.601,Z 598.29,A -85,B 0,C 180,E1 -24008.075,E2 -24008.075} C_VEL
LIN {X 0,Y 152.565,Z 591.515,A -85,B 0,C 180,E1 -24011.841,E2 -24011.841} C_VEL
LIN {X 0,Y 155.084,Z 582.967,A -85,B 0,C 180,E1 -24015.564,E2 -24015.564} C_VEL
LIN {X 0,Y 157.696,Z 573.971,A -85,B 0,C 180,E1 -24018.66,E2 -24018.66} C_VEL
LIN {X 0,Y 160.534,Z 563.547,A -85,B 0,C 180,E1 -24021.5,E2 -24021.5} C_VEL
LIN {X 0,Y 163.172,Z 552.616,A -85,B 0,C 180,E1 -24023.814,E2 -24023.814} C_VEL
LIN {X 0,Y 165.818,Z 539.674,A -85,B 0,C 180,E1 -24025.895,E2 -24025.895} C_VEL
LIN {X 0,Y 167.722,Z 527.893,A -85,B 0,C 180,E1 -24027.295,E2 -24027.295} C_VEL
LIN {X 0,Y 169.223,Z 515.152,A -85,B 0,C 180,E1 -24028.345,E2 -24028.345} C_VEL
LIN {X 0,Y 170.565,Z 497.019,A -85,B 0,C 180,E1 -24029.237,E2 -24029.237} C_VEL
LIN {X 0,Y 172.854,Z 459.787,A -85,B 0,C 180,E1 -24030.855,E2 -24030.855} C_VEL
LIN {X 0,Y 168.39,Z 447.203,A -85,B 0,C 180,E1 -24032.437,E2 -24032.437} C_VEL
LIN {X 0,Y 161.676,Z 432.367,A -85,B 0,C 180,E1 -24034.776,E2 -24034.776} C_VEL
LIN {X 0,Y 152.379,Z 416.387,A -85,B 0,C 180,E1 -24038.109,E2 -24038.109} C_VEL
LIN {X 0,Y 150.896,Z 413.612,A -85,B 0,C 180,E1 -24038.703,E2 -24038.703} C_VEL
LIN {X 0,Y 150.722,Z 412.709,A -85,B 0,C 180,E1 -24038.882,E2 -24038.882} C_VEL
LIN {X 0,Y 150.465,Z 412.735,A -85,B 0,C 180,E1 -24043.502,E2 -24043.502} C_VEL
LIN {X 0,Y 150.367,Z 412.739,A -85,B 0,C 180,E1 -24049.093,E2 -24049.093} C_VEL
LIN {X 0,Y 150.224,Z 412.766,A -85,B 0,C 180,E1 -24054.897,E2 -24054.897} C_VEL
LIN {X 0,Y 150.219,Z 412.749,A -85,B 0,C 180,E1 -24057.891,E2 -24057.891} C_VEL
LIN {X 0,Y 150.266,Z 412.763,A -85,B 0,C 180,E1 -24061.165,E2 -24061.165} C_VEL
LIN {X 0,Y 161.029,Z 442.949,A -85,B 0,C 180,E1 -24064.658,E2 -24064.658} C_VEL
LIN {X 0,Y 163.245,Z 450.6,A -85,B 0,C 180,E1 -24065.4,E2 -24065.4} C_VEL
LIN {X 0,Y 159.031,Z 512.327,A -85,B 0,C 180,E1 -24069.342,E2 -24069.342} C_VEL
LIN {X 0,Y 157.921,Z 525.223,A -85,B 0,C 180,E1 -24070.593,E2 -24070.593} C_VEL
LIN {X 0,Y 156.448,Z 538.125,A -85,B 0,C 180,E1 -24072.359,E2 -24072.359} C_VEL
LIN {X 0,Y 154.857,Z 549.45,A -85,B 0,C 180,E1 -24074.373,E2 -24074.373} C_VEL
LIN {X 0,Y 152.999,Z 561.536,A -85,B 0,C 180,E1 -24077.142,E2 -24077.142} C_VEL
LIN {X 0,Y 151.264,Z 572.412,A -85,B 0,C 180,E1 -24080.293,E2 -24080.293} C_VEL
LIN {X 0,Y 149.782,Z 582.737,A -85,B 0,C 180,E1 -24084.089,E2 -24084.089} C_VEL
LIN {X 0,Y 148.643,Z 591.072,A -85,B 0,C 180,E1 -24087.94,E2 -24087.94} C_VEL
LIN {X 0,Y 148.035,Z 597.564,A -85,B 0,C 180,E1 -24091.656,E2 -24091.656} C_VEL
LIN {X 0,Y 147.451,Z 603.768,A -85,B 0,C 180,E1 -24096.163,E2 -24096.163} C_VEL
LIN {X 0,Y 147.401,Z 608.387,A -85,B 0,C 180,E1 -24100.503,E2 -24100.503} C_VEL
LIN {X 0,Y 147.689,Z 610.822,A -85,B 0,C 180,E1 -24103.41,E2 -24103.41} C_VEL
LIN {X 0,Y 148.284,Z 612.742,A -85,B 0,C 180,E1 -24106.291,E2 -24106.291} C_VEL
LIN {X 0,Y 149.695,Z 614.733,A -85,B 0,C 180,E1 -24110.352,E2 -24110.352} C_VEL
LIN {X 0,Y 151.964,Z 615.894,A -85,B 0,C 180,E1 -24114.693,E2 -24114.693} C_VEL
LIN {X 0,Y 156.232,Z 615.871,A -85,B 0,C 180,E1 -24120,E2 -24120} C_VEL
LIN {X 0,Y 158.835,Z 615.264,A -85,B 0,C 180,E1 -24122.536,E2 -24122.536} C_VEL
LIN {X 0,Y 162.369,Z 613.959,A -85,B 0,C 180,E1 -24125.458,E2 -24125.458} C_VEL
LIN {X 0,Y 168.561,Z 610.857,A -85,B 0,C 180,E1 -24129.6,E2 -24129.6} C_VEL
LIN {X 0,Y 174.477,Z 607.102,A -85,B 0,C 180,E1 -24132.799,E2 -24132.799} C_VEL
LIN {X 0,Y 180.969,Z 602.222,A -85,B 0,C 180,E1 -24135.774,E2 -24135.774} C_VEL
LIN {X 0,Y 189.321,Z 594.748,A -85,B 0,C 180,E1 -24138.954,E2 -24138.954} C_VEL
LIN {X 0,Y 197.05,Z 586.681,A -85,B 0,C 180,E1 -24141.461,E2 -24141.461} C_VEL
LIN {X 0,Y 203.855,Z 578.352,A -85,B 0,C 180,E1 -24143.358,E2 -24143.358} C_VEL
LIN {X 0,Y 211.294,Z 567.712,A -85,B 0,C 180,E1 -24145.256,E2 -24145.256} C_VEL
LIN {X 0,Y 217.432,Z 557.266,A -85,B 0,C 180,E1 -24146.646,E2 -24146.646} C_VEL
LIN {X 0,Y 223.657,Z 544.295,A -85,B 0,C 180,E1 -24147.944,E2 -24147.944} C_VEL
LIN {X 0,Y 227.982,Z 533.194,A -85,B 0,C 180,E1 -24148.753,E2 -24148.753} C_VEL
LIN {X 0,Y 231.683,Z 520.88,A -85,B 0,C 180,E1 -24149.428,E2 -24149.428} C_VEL
LIN {X 0,Y 234.655,Z 507.129,A -85,B 0,C 180,E1 -24149.982,E2 -24149.982} C_VEL
LIN {X 0,Y 234.429,Z 506.088,A -85,B 0,C 180,E1 -24150.935,E2 -24150.935} C_VEL
LIN {X 0,Y 234.1,Z 505.559,A -85,B 0,C 180,E1 -24152.802,E2 -24152.802} C_VEL
LIN {X 0,Y 234.137,Z 505.745,A -85,B 0,C 180,E1 -24155.459,E2 -24155.459} C_VEL
LIN {X 0,Y 234.421,Z 506.768,A -85,B 0,C 180,E1 -24157.11,E2 -24157.11} C_VEL
LIN {X 0,Y 234.557,Z 507.546,A -85,B 0,C 180,E1 -24157.792,E2 -24157.792} C_VEL
LIN {X 0,Y 230.834,Z 524.446,A -85,B 0,C 180,E1 -24158.484,E2 -24158.484} C_VEL
LIN {X 0,Y 226.607,Z 537.647,A -85,B 0,C 180,E1 -24159.167,E2 -24159.167} C_VEL
LIN {X 0,Y 221.412,Z 550.272,A -85,B 0,C 180,E1 -24160.029,E2 -24160.029} C_VEL
LIN {X 0,Y 214.92,Z 562.811,A -85,B 0,C 180,E1 -24161.231,E2 -24161.231} C_VEL
LIN {X 0,Y 212.645,Z 566.655,A -85,B 0,C 180,E1 -24161.68,E2 -24161.68} C_VEL
LIN {X 0,Y 209.478,Z 571.433,A -85,B 0,C 180,E1 -24162.137,E2 -24162.137} C_VEL
LIN {X 0,Y 203.324,Z 579.092,A -85,B 0,C 180,E1 -24162.552,E2 -24162.552} C_VEL
LIN {X 0,Y 196.832,Z 586.195,A -85,B 0,C 180,E1 -24163.112,E2 -24163.112} C_VEL
LIN {X 0,Y 193.174,Z 590.087,A -85,B 0,C 180,E1 -24163.81,E2 -24163.81} C_VEL
LIN {X 0,Y 185.054,Z 598.28,A -85,B 0,C 180,E1 -24166.128,E2 -24166.128} C_VEL
LIN {X 0,Y 176.672,Z 605.546,A -85,B 0,C 180,E1 -24168.981,E2 -24168.981} C_VEL
LIN {X 0,Y 168.451,Z 611.626,A -85,B 0,C 180,E1 -24172.439,E2 -24172.439} C_VEL
LIN {X 0,Y 161.921,Z 615.604,A -85,B 0,C 180,E1 -24175.654,E2 -24175.654} C_VEL
LIN {X 0,Y 155.288,Z 619.101,A -85,B 0,C 180,E1 -24180.147,E2 -24180.147} C_VEL
LIN {X 0,Y 149.592,Z 621.111,A -85,B 0,C 180,E1 -24184.991,E2 -24184.991} C_VEL
LIN {X 0,Y 145.169,Z 621.69,A -85,B 0,C 180,E1 -24190.195,E2 -24190.195} C_VEL
LIN {X 0,Y 142.463,Z 620.879,A -85,B 0,C 180,E1 -24195.724,E2 -24195.724} C_VEL
LIN {X 0,Y 141.181,Z 618.564,A -85,B 0,C 180,E1 -24201.415,E2 -24201.415} C_VEL
LIN {X 0,Y 141.027,Z 617.568,A -85,B 0,C 180,E1 -24203.207,E2 -24203.207} C_VEL
LIN {X 0,Y 140.634,Z 620.904,A -85,B 0,C 180,E1 -24208.139,E2 -24208.139} C_VEL
LIN {X 0,Y 140.594,Z 622.309,A -85,B 0,C 180,E1 -24211.258,E2 -24211.258} C_VEL
LIN {X 0,Y 140.621,Z 623.481,A -85,B 0,C 180,E1 -24215.74,E2 -24215.74} C_VEL
LIN {X 0,Y 141.443,Z 623.595,A -85,B 0,C 180,E1 -24221.468,E2 -24221.468} C_VEL
LIN {X 0,Y 142.317,Z 623.076,A -85,B 0,C 180,E1 -24224.299,E2 -24224.299} C_VEL
LIN {X 0,Y 145.028,Z 620.832,A -85,B 0,C 180,E1 -24229.833,E2 -24229.833} C_VEL
LIN {X 0,Y 148.117,Z 618.122,A -85,B 0,C 180,E1 -24233.789,E2 -24233.789} C_VEL
LIN {X 0,Y 151.755,Z 614.454,A -85,B 0,C 180,E1 -24237.592,E2 -24237.592} C_VEL
LIN {X 0,Y 156.646,Z 609.003,A -85,B 0,C 180,E1 -24241.674,E2 -24241.674} C_VEL
LIN {X 0,Y 161.835,Z 602.707,A -85,B 0,C 180,E1 -24245.132,E2 -24245.132} C_VEL
LIN {X 0,Y 167.39,Z 595.185,A -85,B 0,C 180,E1 -24248.268,E2 -24248.268} C_VEL
LIN {X 0,Y 173.667,Z 585.829,A -85,B 0,C 180,E1 -24251.121,E2 -24251.121} C_VEL
LIN {X 0,Y 179.125,Z 576.302,A -85,B 0,C 180,E1 -24253.366,E2 -24253.366} C_VEL
LIN {X 0,Y 184.362,Z 565.796,A -85,B 0,C 180,E1 -24255.238,E2 -24255.238} C_VEL
LIN {X 0,Y 189.216,Z 554.044,A -85,B 0,C 180,E1 -24256.8,E2 -24256.8} C_VEL
LIN {X 0,Y 193.33,Z 541.724,A -85,B 0,C 180,E1 -24257.987,E2 -24257.987} C_VEL
LIN {X 0,Y 196.648,Z 528.683,A -85,B 0,C 180,E1 -24258.856,E2 -24258.856} C_VEL
LIN {X 0,Y 198.855,Z 514.749,A -85,B 0,C 180,E1 -24259.521,E2 -24259.521} C_VEL
LIN {X 0,Y 201.254,Z 491.514,A -85,B 0,C 180,E1 -24260.366,E2 -24260.366} C_VEL
LIN {X 0,Y 199.117,Z 485.342,A -85,B 0,C 180,E1 -24262.272,E2 -24262.272} C_VEL
LIN {X 0,Y 196.555,Z 478.899,A -85,B 0,C 180,E1 -24264.766,E2 -24264.766} C_VEL
LIN {X 0,Y 193.936,Z 472.905,A -85,B 0,C 180,E1 -24267.776,E2 -24267.776} C_VEL
LIN {X 0,Y 192.106,Z 468.974,A -85,B 0,C 180,E1 -24270.418,E2 -24270.418} C_VEL
LIN {X 0,Y 189.953,Z 464.301,A -85,B 0,C 180,E1 -24274.849,E2 -24274.849} C_VEL
LIN {X 0,Y 188.807,Z 462.288,A -85,B 0,C 180,E1 -24279.931,E2 -24279.931} C_VEL
LIN {X 0,Y 189.043,Z 462.036,A -85,B 0,C 180,E1 -24283.899,E2 -24283.899} C_VEL
LIN {X 0,Y 190.116,Z 463.038,A -85,B 0,C 180,E1 -24287.591,E2 -24287.591} C_VEL
LIN {X 0,Y 191.943,Z 466.245,A -85,B 0,C 180,E1 -24291.358,E2 -24291.358} C_VEL
LIN {X 0,Y 192.948,Z 467.521,A -85,B 0,C 180,E1 -24292.803,E2 -24292.803} C_VEL
LIN {X 0,Y 194.693,Z 470.584,A -85,B 0,C 180,E1 -24295.088,E2 -24295.088} C_VEL
LIN {X 0,Y 197.898,Z 477.064,A -85,B 0,C 180,E1 -24298.516,E2 -24298.516} C_VEL
LIN {X 0,Y 201.281,Z 485.197,A -85,B 0,C 180,E1 -24301.533,E2 -24301.533} C_VEL
LIN {X 0,Y 201.752,Z 486.451,A -85,B 0,C 180,E1 -24301.93,E2 -24301.93} C_VEL
LIN {X 0,Y 198.506,Z 515.497,A -85,B 0,C 180,E1 -24302.98,E2 -24302.98} C_VEL
LIN {X 0,Y 195.967,Z 528.625,A -85,B 0,C 180,E1 -24303.731,E2 -24303.731} C_VEL
LIN {X 0,Y 192.699,Z 540.887,A -85,B 0,C 180,E1 -24304.777,E2 -24304.777} C_VEL
LIN {X 0,Y 188.816,Z 552.049,A -85,B 0,C 180,E1 -24306.054,E2 -24306.054} C_VEL
LIN {X 0,Y 183.867,Z 563.657,A -85,B 0,C 180,E1 -24307.829,E2 -24307.829} C_VEL
LIN {X 0,Y 178.404,Z 574.266,A -85,B 0,C 180,E1 -24309.974,E2 -24309.974} C_VEL
LIN {X 0,Y 172.742,Z 583.573,A -85,B 0,C 180,E1 -24312.45,E2 -24312.45} C_VEL
LIN {X 0,Y 167.457,Z 591.253,A -85,B 0,C 180,E1 -24315.13,E2 -24315.13} C_VEL
LIN {X 0,Y 161.379,Z 599.022,A -85,B 0,C 180,E1 -24318.694,E2 -24318.694} C_VEL
LIN {X 0,Y 155.971,Z 605.051,A -85,B 0,C 180,E1 -24322.516,E2 -24322.516} C_VEL
LIN {X 0,Y 152.112,Z 608.933,A -85,B 0,C 180,E1 -24325.837,E2 -24325.837} C_VEL
LIN {X 0,Y 147.471,Z 613.005,A -85,B 0,C 180,E1 -24330.921,E2 -24330.921} C_VEL
LIN {X 0,Y 144.313,Z 615.285,A -85,B 0,C 180,E1 -24335.761,E2 -24335.761} C_VEL
LIN {X 0,Y 142.341,Z 616.19,A -85,B 0,C 180,E1 -24339.932,E2 -24339.932} C_VEL
LIN {X 0,Y 140.658,Z 616.038,A -85,B 0,C 180,E1 -24345.607,E2 -24345.607} C_VEL
LIN {X 0,Y 140.155,Z 615.119,A -85,B 0,C 180,E1 -24349.312,E2 -24349.312} C_VEL
LIN {X 0,Y 140.03,Z 613.296,A -85,B 0,C 180,E1 -24353.421,E2 -24353.421} C_VEL
LIN {X 0,Y 140.588,Z 610.108,A -85,B 0,C 180,E1 -24358.194,E2 -24358.194} C_VEL
LIN {X 0,Y 141.774,Z 604.978,A -85,B 0,C 180,E1 -24363.499,E2 -24363.499} C_VEL
LIN {X 0,Y 143.569,Z 598.406,A -85,B 0,C 180,E1 -24368.45,E2 -24368.45} C_VEL
LIN {X 0,Y 145.65,Z 591.505,A -85,B 0,C 180,E1 -24372.444,E2 -24372.444} C_VEL
LIN {X 0,Y 148.244,Z 583.008,A -85,B 0,C 180,E1 -24376.285,E2 -24376.285} C_VEL
LIN {X 0,Y 151.072,Z 573.651,A -85,B 0,C 180,E1 -24379.611,E2 -24379.611} C_VEL
LIN {X 0,Y 154.082,Z 562.949,A -85,B 0,C 180,E1 -24382.591,E2 -24382.591} C_VEL
LIN {X 0,Y 157.138,Z 550.666,A -85,B 0,C 180,E1 -24385.186,E2 -24385.186} C_VEL
LIN {X 0,Y 159.663,Z 538.327,A -85,B 0,C 180,E1 -24387.158,E2 -24387.158} C_VEL
LIN {X 0,Y 161.688,Z 525.095,A -85,B 0,C 180,E1 -24388.684,E2 -24388.684} C_VEL
LIN {X 0,Y 163.304,Z 511.436,A -85,B 0,C 180,E1 -24389.713,E2 -24389.713} C_VEL
LIN {X 0,Y 166.662,Z 461.402,A -85,B 0,C 180,E1 -24391.974,E2 -24391.974} C_VEL
LIN {X 0,Y 162.546,Z 449.894,A -85,B 0,C 180,E1 -24393.527,E2 -24393.527} C_VEL
LIN {X 0,Y 156.392,Z 436.27,A -85,B 0,C 180,E1 -24395.779,E2 -24395.779} C_VEL
LIN {X 0,Y 146.745,Z 419.635,A -85,B 0,C 180,E1 -24399.456,E2 -24399.456} C_VEL
LIN {X 0,Y 145.371,Z 417.402,A -85,B 0,C 180,E1 -24400.017,E2 -24400.017} C_VEL
LIN {X 0,Y 143.916,Z 414.828,A -85,B 0,C 180,E1 -24400.642,E2 -24400.642} C_VEL
LIN {X 0,Y 143.644,Z 413.591,A -85,B 0,C 180,E1 -24400.836,E2 -24400.836} C_VEL
LIN {X 0,Y 143.317,Z 413.629,A -85,B 0,C 180,E1 -24407.107,E2 -24407.107} C_VEL
LIN {X 0,Y 143.276,Z 413.632,A -85,B 0,C 180,E1 -24411.251,E2 -24411.251} C_VEL
LIN {X 0,Y 143.188,Z 413.624,A -85,B 0,C 180,E1 -24417.933,E2 -24417.933} C_VEL
LIN {X 0,Y 143.171,Z 413.641,A -85,B 0,C 180,E1 -24420.306,E2 -24420.306} C_VEL
LIN {X 0,Y 154.433,Z 445.11,A -85,B 0,C 180,E1 -24424.117,E2 -24424.117} C_VEL
LIN {X 0,Y 156.351,Z 451.678,A -85,B 0,C 180,E1 -24424.794,E2 -24424.794} C_VEL
LIN {X 0,Y 151.999,Z 513.18,A -85,B 0,C 180,E1 -24428.915,E2 -24428.915} C_VEL
LIN {X 0,Y 150.927,Z 525.252,A -85,B 0,C 180,E1 -24430.149,E2 -24430.149} C_VEL
LIN {X 0,Y 149.277,Z 539.09,A -85,B 0,C 180,E1 -24432.139,E2 -24432.139} C_VEL
LIN {X 0,Y 147.575,Z 551.004,A -85,B 0,C 180,E1 -24434.409,E2 -24434.409} C_VEL
LIN {X 0,Y 145.891,Z 561.522,A -85,B 0,C 180,E1 -24436.98,E2 -24436.98} C_VEL
LIN {X 0,Y 144.163,Z 572.163,A -85,B 0,C 180,E1 -24440.219,E2 -24440.219} C_VEL
LIN {X 0,Y 142.794,Z 581.588,A -85,B 0,C 180,E1 -24443.799,E2 -24443.799} C_VEL
LIN {X 0,Y 141.556,Z 590.672,A -85,B 0,C 180,E1 -24448.115,E2 -24448.115} C_VEL
LIN {X 0,Y 140.983,Z 596.829,A -85,B 0,C 180,E1 -24451.733,E2 -24451.733} C_VEL
LIN {X 0,Y 140.518,Z 601.717,A -85,B 0,C 180,E1 -24455.222,E2 -24455.222} C_VEL
LIN {X 0,Y 140.306,Z 606.498,A -85,B 0,C 180,E1 -24459.474,E2 -24459.474} C_VEL
LIN {X 0,Y 140.716,Z 610.491,A -85,B 0,C 180,E1 -24464.056,E2 -24464.056} C_VEL
LIN {X 0,Y 141.844,Z 613.381,A -85,B 0,C 180,E1 -24468.569,E2 -24468.569} C_VEL
LIN {X 0,Y 143.018,Z 614.747,A -85,B 0,C 180,E1 -24471.522,E2 -24471.522} C_VEL
LIN {X 0,Y 144.5,Z 615.688,A -85,B 0,C 180,E1 -24474.418,E2 -24474.418} C_VEL
LIN {X 0,Y 148.718,Z 616.314,A -85,B 0,C 180,E1 -24480,E2 -24480} C_VEL
LIN {X 0,Y 151.362,Z 616.039,A -85,B 0,C 180,E1 -24482.661,E2 -24482.661} C_VEL
LIN {X 0,Y 155.503,Z 614.954,A -85,B 0,C 180,E1 -24486.16,E2 -24486.16} C_VEL
LIN {X 0,Y 161.228,Z 612.661,A -85,B 0,C 180,E1 -24490.041,E2 -24490.041} C_VEL
LIN {X 0,Y 167.43,Z 609.402,A -85,B 0,C 180,E1 -24493.458,E2 -24493.458} C_VEL
LIN {X 0,Y 173.892,Z 605.233,A -85,B 0,C 180,E1 -24496.434,E2 -24496.434} C_VEL
LIN {X 0,Y 181.148,Z 599.77,A -85,B 0,C 180,E1 -24499.255,E2 -24499.255} C_VEL
LIN {X 0,Y 188.933,Z 592.821,A -85,B 0,C 180,E1 -24501.838,E2 -24501.838} C_VEL
LIN {X 0,Y 197.157,Z 584.247,A -85,B 0,C 180,E1 -24504.201,E2 -24504.201} C_VEL
LIN {X 0,Y 204.954,Z 574.646,A -85,B 0,C 180,E1 -24506.135,E2 -24506.135} C_VEL
LIN {X 0,Y 212.583,Z 563.426,A -85,B 0,C 180,E1 -24507.828,E2 -24507.828} C_VEL
LIN {X 0,Y 218.826,Z 552.401,A -85,B 0,C 180,E1 -24509.063,E2 -24509.063} C_VEL
LIN {X 0,Y 224.287,Z 540.508,A -85,B 0,C 180,E1 -24510.09,E2 -24510.09} C_VEL
LIN {X 0,Y 229.019,Z 527.384,A -85,B 0,C 180,E1 -24510.894,E2 -24510.894} C_VEL
LIN {X 0,Y 232.706,Z 513.494,A -85,B 0,C 180,E1 -24511.489,E2 -24511.489} C_VEL
LIN {X 0,Y 232.839,Z 512.799,A -85,B 0,C 180,E1 -24511.561,E2 -24511.561} C_VEL
LIN {X 0,Y 232.619,Z 512.505,A -85,B 0,C 180,E1 -24512.944,E2 -24512.944} C_VEL
LIN {X 0,Y 232.692,Z 512.829,A -85,B 0,C 180,E1 -24515.713,E2 -24515.713} C_VEL
LIN {X 0,Y 232.766,Z 513.082,A -85,B 0,C 180,E1 -24516.265,E2 -24516.265} C_VEL
LIN {X 0,Y 229.168,Z 527.307,A -85,B 0,C 180,E1 -24516.838,E2 -24516.838} C_VEL
LIN {X 0,Y 224.555,Z 540.467,A -85,B 0,C 180,E1 -24517.532,E2 -24517.532} C_VEL
LIN {X 0,Y 218.685,Z 553.308,A -85,B 0,C 180,E1 -24518.436,E2 -24518.436} C_VEL
LIN {X 0,Y 211.99,Z 565.195,A -85,B 0,C 180,E1 -24519.579,E2 -24519.579} C_VEL
LIN {X 0,Y 204.905,Z 575.793,A -85,B 0,C 180,E1 -24521.016,E2 -24521.016} C_VEL
LIN {X 0,Y 198.034,Z 584.564,A -85,B 0,C 180,E1 -24522.579,E2 -24522.579} C_VEL
LIN {X 0,Y 193.174,Z 590.087,A -85,B 0,C 180,E1 -24523.81,E2 -24523.81} C_VEL
LIN {X 0,Y 189.361,Z 593.871,A -85,B 0,C 180,E1 -24524.588,E2 -24524.588} C_VEL
LIN {X 0,Y 182.017,Z 599.838,A -85,B 0,C 180,E1 -24525.546,E2 -24525.546} C_VEL
LIN {X 0,Y 174.52,Z 605.079,A -85,B 0,C 180,E1 -24526.701,E2 -24526.701} C_VEL
LIN {X 0,Y 170.537,Z 607.754,A -85,B 0,C 180,E1 -24527.802,E2 -24527.802} C_VEL
LIN {X 0,Y 163.656,Z 612.295,A -85,B 0,C 180,E1 -24530.623,E2 -24530.623} C_VEL
LIN {X 0,Y 156.145,Z 616.377,A -85,B 0,C 180,E1 -24534.193,E2 -24534.193} C_VEL
LIN {X 0,Y 149.179,Z 619.435,A -85,B 0,C 180,E1 -24538.791,E2 -24538.791} C_VEL
LIN {X 0,Y 143.177,Z 621.126,A -85,B 0,C 180,E1 -24543.787,E2 -24543.787} C_VEL
LIN {X 0,Y 138.504,Z 621.395,A -85,B 0,C 180,E1 -24549.199,E2 -24549.199} C_VEL
LIN {X 0,Y 135.601,Z 620.239,A -85,B 0,C 180,E1 -24554.985,E2 -24554.985} C_VEL
LIN {X 0,Y 134.218,Z 617.673,A -85,B 0,C 180,E1 -24560.966,E2 -24560.966} C_VEL
LIN {X 0,Y 134.037,Z 616.751,A -85,B 0,C 180,E1 -24562.661,E2 -24562.661} C_VEL
LIN {X 0,Y 133.569,Z 620.715,A -85,B 0,C 180,E1 -24568.647,E2 -24568.647} C_VEL
LIN {X 0,Y 133.466,Z 622.488,A -85,B 0,C 180,E1 -24573.022,E2 -24573.022} C_VEL
LIN {X 0,Y 133.548,Z 623.187,A -85,B 0,C 180,E1 -24576.045,E2 -24576.045} C_VEL
LIN {X 0,Y 134.479,Z 623.42,A -85,B 0,C 180,E1 -24582.07,E2 -24582.07} C_VEL
LIN {X 0,Y 136.681,Z 622.158,A -85,B 0,C 180,E1 -24587.974,E2 -24587.974} C_VEL
LIN {X 0,Y 140.464,Z 619.297,A -85,B 0,C 180,E1 -24593.599,E2 -24593.599} C_VEL
LIN {X 0,Y 144.176,Z 616.086,A -85,B 0,C 180,E1 -24597.59,E2 -24597.59} C_VEL
LIN {X 0,Y 149.469,Z 610.816,A -85,B 0,C 180,E1 -24602.183,E2 -24602.183} C_VEL
LIN {X 0,Y 155.2,Z 604.55,A -85,B 0,C 180,E1 -24606.068,E2 -24606.068} C_VEL
LIN {X 0,Y 160.968,Z 597.486,A -85,B 0,C 180,E1 -24609.282,E2 -24609.282} C_VEL
LIN {X 0,Y 167.353,Z 588.761,A -85,B 0,C 180,E1 -24612.219,E2 -24612.219} C_VEL
LIN {X 0,Y 172.943,Z 579.917,A -85,B 0,C 180,E1 -24614.511,E2 -24614.511} C_VEL
LIN {X 0,Y 178.91,Z 569.041,A -85,B 0,C 180,E1 -24616.616,E2 -24616.616} C_VEL
LIN {X 0,Y 184.535,Z 556.746,A -85,B 0,C 180,E1 -24618.371,E2 -24618.371} C_VEL
LIN {X 0,Y 188.438,Z 546.354,A -85,B 0,C 180,E1 -24619.46,E2 -24619.46} C_VEL
LIN {X 0,Y 192.126,Z 533.978,A -85,B 0,C 180,E1 -24620.403,E2 -24620.403} C_VEL
LIN {X 0,Y 195.034,Z 519.685,A -85,B 0,C 180,E1 -24621.171,E2 -24621.171} C_VEL
LIN {X 0,Y 197.877,Z 494.571,A -85,B 0,C 180,E1 -24622.105,E2 -24622.105} C_VEL
LIN {X 0,Y 195.423,Z 487.585,A -85,B 0,C 180,E1 -24624.574,E2 -24624.574} C_VEL
LIN {X 0,Y 193.294,Z 482.089,A -85,B 0,C 180,E1 -24627.052,E2 -24627.052} C_VEL
LIN {X 0,Y 192.007,Z 478.947,A -85,B 0,C 180,E1 -24628.779,E2 -24628.779} C_VEL
LIN {X 0,Y 190.523,Z 475.44,A -85,B 0,C 180,E1 -24631.163,E2 -24631.163} C_VEL
LIN {X 0,Y 188.738,Z 471.171,A -85,B 0,C 180,E1 -24635.242,E2 -24635.242} C_VEL
LIN {X 0,Y 187.765,Z 469.368,A -85,B 0,C 180,E1 -24639.815,E2 -24639.815} C_VEL
LIN {X 0,Y 187.81,Z 468.969,A -85,B 0,C 180,E1 -24642.581,E2 -24642.581} C_VEL
LIN {X 0,Y 188.87,Z 469.815,A -85,B 0,C 180,E1 -24647.099,E2 -24647.099} C_VEL
LIN {X 0,Y 190.609,Z 473.097,A -85,B 0,C 180,E1 -24650.984,E2 -24650.984} C_VEL
LIN {X 0,Y 191.483,Z 474.325,A -85,B 0,C 180,E1 -24652.315,E2 -24652.315} C_VEL
LIN {X 0,Y 192.977,Z 477.183,A -85,B 0,C 180,E1 -24654.44,E2 -24654.44} C_VEL
LIN {X 0,Y 195.806,Z 483.262,A -85,B 0,C 180,E1 -24657.682,E2 -24657.682} C_VEL
LIN {X 0,Y 198.326,Z 489.816,A -85,B 0,C 180,E1 -24660.183,E2 -24660.183} C_VEL
LIN {X 0,Y 195.256,Z 516.195,A -85,B 0,C 180,E1 -24661.155,E2 -24661.155} C_VEL
LIN {X 0,Y 192.567,Z 529.47,A -85,B 0,C 180,E1 -24661.914,E2 -24661.914} C_VEL
LIN {X 0,Y 188.816,Z 542.478,A -85,B 0,C 180,E1 -24663.034,E2 -24663.034} C_VEL
LIN {X 0,Y 184.607,Z 553.791,A -85,B 0,C 180,E1 -24664.367,E2 -24664.367} C_VEL
LIN {X 0,Y 179.378,Z 565.246,A -85,B 0,C 180,E1 -24666.168,E2 -24666.168} C_VEL
LIN {X 0,Y 173.968,Z 575.066,A -85,B 0,C 180,E1 -24668.19,E2 -24668.19} C_VEL
LIN {X 0,Y 168.069,Z 584.273,A -85,B 0,C 180,E1 -24670.665,E2 -24670.665} C_VEL
LIN {X 0,Y 162.526,Z 591.855,A -85,B 0,C 180,E1 -24673.344,E2 -24673.344} C_VEL
LIN {X 0,Y 156.805,Z 598.748,A -85,B 0,C 180,E1 -24676.535,E2 -24676.535} C_VEL
LIN {X 0,Y 151.827,Z 604.01,A -85,B 0,C 180,E1 -24679.752,E2 -24679.752} C_VEL
LIN {X 0,Y 146.349,Z 609.201,A -85,B 0,C 180,E1 -24684.151,E2 -24684.151} C_VEL
LIN {X 0,Y 142.795,Z 612.142,A -85,B 0,C 180,E1 -24687.629,E2 -24687.629} C_VEL
LIN {X 0,Y 139.828,Z 614.276,A -85,B 0,C 180,E1 -24691.295,E2 -24691.295} C_VEL
LIN {X 0,Y 137.424,Z 615.703,A -85,B 0,C 180,E1 -24695.084,E2 -24695.084} C_VEL
LIN {X 0,Y 135.561,Z 616.437,A -85,B 0,C 180,E1 -24698.948,E2 -24698.948} C_VEL
LIN {X 0,Y 134.21,Z 616.453,A -85,B 0,C 180,E1 -24702.903,E2 -24702.903} C_VEL
LIN {X 0,Y 133.208,Z 615.611,A -85,B 0,C 180,E1 -24707.616,E2 -24707.616} C_VEL
LIN {X 0,Y 132.906,Z 613.727,A -85,B 0,C 180,E1 -24712.485,E2 -24712.485} C_VEL
LIN {X 0,Y 133.5,Z 610.117,A -85,B 0,C 180,E1 -24718.23,E2 -24718.23} C_VEL
LIN {X 0,Y 134.437,Z 606.08,A -85,B 0,C 180,E1 -24722.713,E2 -24722.713} C_VEL
LIN {X 0,Y 135.75,Z 601.147,A -85,B 0,C 180,E1 -24726.934,E2 -24726.934} C_VEL
LIN {X 0,Y 137.812,Z 594.436,A -85,B 0,C 180,E1 -24731.41,E2 -24731.41} C_VEL
LIN {X 0,Y 140.276,Z 586.594,A -85,B 0,C 180,E1 -24735.489,E2 -24735.489} C_VEL
LIN {X 0,Y 143.13,Z 577.694,A -85,B 0,C 180,E1 -24739.129,E2 -24739.129} C_VEL
LIN {X 0,Y 146.262,Z 567.49,A -85,B 0,C 180,E1 -24742.388,E2 -24742.388} C_VEL
LIN {X 0,Y 149.462,Z 555.687,A -85,B 0,C 180,E1 -24745.276,E2 -24745.276} C_VEL
LIN {X 0,Y 152.024,Z 544.691,A -85,B 0,C 180,E1 -24747.347,E2 -24747.347} C_VEL
LIN {X 0,Y 154.421,Z 532.135,A -85,B 0,C 180,E1 -24749.108,E2 -24749.108} C_VEL
LIN {X 0,Y 156.234,Z 519.459,A -85,B 0,C 180,E1 -24750.368,E2 -24750.368} C_VEL
LIN {X 0,Y 157.505,Z 506.74,A -85,B 0,C 180,E1 -24751.177,E2 -24751.177} C_VEL
LIN {X 0,Y 160.463,Z 462.893,A -85,B 0,C 180,E1 -24753.204,E2 -24753.204} C_VEL
LIN {X 0,Y 157.223,Z 453.823,A -85,B 0,C 180,E1 -24754.475,E2 -24754.475} C_VEL
LIN {X 0,Y 151.242,Z 440.278,A -85,B 0,C 180,E1 -24756.811,E2 -24756.811} C_VEL
LIN {X 0,Y 141.004,Z 422.422,A -85,B 0,C 180,E1 -24760.993,E2 -24760.993} C_VEL
LIN {X 0,Y 138.53,Z 418.611,A -85,B 0,C 180,E1 -24762.081,E2 -24762.081} C_VEL
LIN {X 0,Y 136.932,Z 416.409,A -85,B 0,C 180,E1 -24762.793,E2 -24762.793} C_VEL
LIN {X 0,Y 136.384,Z 414.487,A -85,B 0,C 180,E1 -24763.234,E2 -24763.234} C_VEL
LIN {X 0,Y 136.252,Z 414.5,A -85,B 0,C 180,E1 -24768.024,E2 -24768.024} C_VEL
LIN {X 0,Y 136.197,Z 414.516,A -85,B 0,C 180,E1 -24771.745,E2 -24771.745} C_VEL
LIN {X 0,Y 136.12,Z 414.508,A -85,B 0,C 180,E1 -24779.021,E2 -24779.021} C_VEL
LIN {X 0,Y 136.103,Z 414.513,A -85,B 0,C 180,E1 -24779.365,E2 -24779.365} C_VEL
LIN {X 0,Y 147.771,Z 446.972,A -85,B 0,C 180,E1 -24783.508,E2 -24783.508} C_VEL
LIN {X 0,Y 149.432,Z 452.677,A -85,B 0,C 180,E1 -24784.131,E2 -24784.131} C_VEL
LIN {X 0,Y 145.07,Z 512.604,A -85,B 0,C 180,E1 -24788.351,E2 -24788.351} C_VEL
LIN {X 0,Y 143.914,Z 525.447,A -85,B 0,C 180,E1 -24789.722,E2 -24789.722} C_VEL
LIN {X 0,Y 142.151,Z 539.542,A -85,B 0,C 180,E1 -24791.866,E2 -24791.866} C_VEL
LIN {X 0,Y 140.506,Z 550.916,A -85,B 0,C 180,E1 -24794.155,E2 -24794.155} C_VEL
LIN {X 0,Y 138.526,Z 562.916,A -85,B 0,C 180,E1 -24797.267,E2 -24797.267} C_VEL
LIN {X 0,Y 136.87,Z 573.101,A -85,B 0,C 180,E1 -24800.59,E2 -24800.59} C_VEL
LIN {X 0,Y 135.524,Z 582.257,A -85,B 0,C 180,E1 -24804.309,E2 -24804.309} C_VEL
LIN {X 0,Y 134.434,Z 590.554,A -85,B 0,C 180,E1 -24808.48,E2 -24808.48} C_VEL
LIN {X 0,Y 133.81,Z 597.372,A -85,B 0,C 180,E1 -24812.738,E2 -24812.738} C_VEL
LIN {X 0,Y 133.342,Z 602.501,A -85,B 0,C 180,E1 -24816.715,E2 -24816.715} C_VEL
LIN {X 0,Y 133.356,Z 607.519,A -85,B 0,C 180,E1 -24821.566,E2 -24821.566} C_VEL
LIN {X 0,Y 134.063,Z 611.27,A -85,B 0,C 180,E1 -24826.355,E2 -24826.355} C_VEL
LIN {X 0,Y 135.63,Z 613.968,A -85,B 0,C 180,E1 -24831.057,E2 -24831.057} C_VEL
LIN {X 0,Y 137.061,Z 615.231,A -85,B 0,C 180,E1 -24834.114,E2 -24834.114} C_VEL
LIN {X 0,Y 141.231,Z 616.501,A -85,B 0,C 180,E1 -24840,E2 -24840} C_VEL
LIN {X 0,Y 143.855,Z 616.554,A -85,B 0,C 180,E1 -24842.8,E2 -24842.8} C_VEL
LIN {X 0,Y 148.669,Z 615.798,A -85,B 0,C 180,E1 -24846.947,E2 -24846.947} C_VEL
LIN {X 0,Y 153.878,Z 614.211,A -85,B 0,C 180,E1 -24850.526,E2 -24850.526} C_VEL
LIN {X 0,Y 158.946,Z 612.113,A -85,B 0,C 180,E1 -24853.421,E2 -24853.421} C_VEL
LIN {X 0,Y 166.784,Z 607.984,A -85,B 0,C 180,E1 -24857.156,E2 -24857.156} C_VEL
LIN {X 0,Y 174.166,Z 603.2,A -85,B 0,C 180,E1 -24860.059,E2 -24860.059} C_VEL
LIN {X 0,Y 183.289,Z 596.127,A -85,B 0,C 180,E1 -24863.046,E2 -24863.046} C_VEL
LIN {X 0,Y 191.943,Z 588.076,A -85,B 0,C 180,E1 -24865.482,E2 -24865.482} C_VEL
LIN {X 0,Y 200.946,Z 578.131,A -85,B 0,C 180,E1 -24867.608,E2 -24867.608} C_VEL
LIN {X 0,Y 208.585,Z 568.041,A -85,B 0,C 180,E1 -24869.231,E2 -24869.231} C_VEL
LIN {X 0,Y 215.802,Z 556.513,A -85,B 0,C 180,E1 -24870.588,E2 -24870.588} C_VEL
LIN {X 0,Y 221.804,Z 544.929,A -85,B 0,C 180,E1 -24871.628,E2 -24871.628} C_VEL
LIN {X 0,Y 226.81,Z 532.742,A -85,B 0,C 180,E1 -24872.4,E2 -24872.4} C_VEL
LIN {X 0,Y 230.946,Z 519.411,A -85,B 0,C 180,E1 -24873.046,E2 -24873.046} C_VEL
LIN {X 0,Y 230.938,Z 519.592,A -85,B 0,C 180,E1 -24874.752,E2 -24874.752} C_VEL
LIN {X 0,Y 226.583,Z 533.543,A -85,B 0,C 180,E1 -24875.324,E2 -24875.324} C_VEL
LIN {X 0,Y 221.579,Z 545.669,A -85,B 0,C 180,E1 -24876.026,E2 -24876.026} C_VEL
LIN {X 0,Y 215.366,Z 557.784,A -85,B 0,C 180,E1 -24876.922,E2 -24876.922} C_VEL
LIN {X 0,Y 208.527,Z 568.775,A -85,B 0,C 180,E1 -24878.023,E2 -24878.023} C_VEL
LIN {X 0,Y 201.991,Z 577.674,A -85,B 0,C 180,E1 -24879.276,E2 -24879.276} C_VEL
LIN {X 0,Y 193.503,Z 587.612,A -85,B 0,C 180,E1 -24881.101,E2 -24881.101} C_VEL
LIN {X 0,Y 185.341,Z 595.764,A -85,B 0,C 180,E1 -24883.126,E2 -24883.126} C_VEL
LIN {X 0,Y 176.363,Z 603.428,A -85,B 0,C 180,E1 -24885.788,E2 -24885.788} C_VEL
LIN {X 0,Y 170.537,Z 607.754,A -85,B 0,C 180,E1 -24887.802,E2 -24887.802} C_VEL
LIN {X 0,Y 166.493,Z 610.302,A -85,B 0,C 180,E1 -24889.015,E2 -24889.015} C_VEL
LIN {X 0,Y 155.525,Z 615.304,A -85,B 0,C 180,E1 -24891.481,E2 -24891.481} C_VEL
LIN {X 0,Y 149.73,Z 617.453,A -85,B 0,C 180,E1 -24893.293,E2 -24893.293} C_VEL
LIN {X 0,Y 147.428,Z 618.263,A -85,B 0,C 180,E1 -24894.455,E2 -24894.455} C_VEL
LIN {X 0,Y 143.165,Z 619.753,A -85,B 0,C 180,E1 -24897.322,E2 -24897.322} C_VEL
LIN {X 0,Y 136.832,Z 621.054,A -85,B 0,C 180,E1 -24902.472,E2 -24902.472} C_VEL
LIN {X 0,Y 131.889,Z 620.986,A -85,B 0,C 180,E1 -24908.103,E2 -24908.103} C_VEL
LIN {X 0,Y 128.767,Z 619.565,A -85,B 0,C 180,E1 -24914.168,E2 -24914.168} C_VEL
LIN {X 0,Y 127.266,Z 616.666,A -85,B 0,C 180,E1 -24920.468,E2 -24920.468} C_VEL
LIN {X 0,Y 127.065,Z 615.927,A -85,B 0,C 180,E1 -24922.056,E2 -24922.056} C_VEL
LIN {X 0,Y 126.499,Z 619.245,A -85,B 0,C 180,E1 -24926.819,E2 -24926.819} C_VEL
LIN {X 0,Y 126.506,Z 621.02,A -85,B 0,C 180,E1 -24930.326,E2 -24930.326} C_VEL
LIN {X 0,Y 126.5,Z 622.875,A -85,B 0,C 180,E1 -24936.384,E2 -24936.384} C_VEL
LIN {X 0,Y 127.51,Z 623.248,A -85,B 0,C 180,E1 -24942.741,E2 -24942.741} C_VEL
LIN {X 0,Y 129.915,Z 622.128,A -85,B 0,C 180,E1 -24948.944,E2 -24948.944} C_VEL
LIN {X 0,Y 131.757,Z 621.007,A -85,B 0,C 180,E1 -24951.928,E2 -24951.928} C_VEL
LIN {X 0,Y 136.55,Z 617.505,A -85,B 0,C 180,E1 -24957.599,E2 -24957.599} C_VEL
LIN {X 0,Y 140.87,Z 613.803,A -85,B 0,C 180,E1 -24961.595,E2 -24961.595} C_VEL
LIN {X 0,Y 145.84,Z 609.057,A -85,B 0,C 180,E1 -24965.333,E2 -24965.333} C_VEL
LIN {X 0,Y 152.578,Z 602.002,A -85,B 0,C 180,E1 -24969.302,E2 -24969.302} C_VEL
LIN {X 0,Y 157.722,Z 595.79,A -85,B 0,C 180,E1 -24971.947,E2 -24971.947} C_VEL
LIN {X 0,Y 164.547,Z 586.789,A -85,B 0,C 180,E1 -24974.812,E2 -24974.812} C_VEL
LIN {X 0,Y 171.104,Z 576.545,A -85,B 0,C 180,E1 -24977.244,E2 -24977.244} C_VEL
LIN {X 0,Y 176.773,Z 566.226,A -85,B 0,C 180,E1 -24979.063,E2 -24979.063} C_VEL
LIN {X 0,Y 181.999,Z 554.832,A -85,B 0,C 180,E1 -24980.566,E2 -24980.566} C_VEL
LIN {X 0,Y 186.392,Z 542.894,A -85,B 0,C 180,E1 -24981.701,E2 -24981.701} C_VEL
LIN {X 0,Y 190.158,Z 529.575,A -85,B 0,C 180,E1 -24982.581,E2 -24982.581} C_VEL
LIN {X 0,Y 192.589,Z 516.184,A -85,B 0,C 180,E1 -24983.229,E2 -24983.229} C_VEL
LIN {X 0,Y 194.683,Z 497.933,A -85,B 0,C 180,E1 -24983.888,E2 -24983.888} C_VEL
LIN {X 0,Y 192.37,Z 490.842,A -85,B 0,C 180,E1 -24986.653,E2 -24986.653} C_VEL
LIN {X 0,Y 190.384,Z 485.446,A -85,B 0,C 180,E1 -24989.464,E2 -24989.464} C_VEL
LIN {X 0,Y 188.902,Z 481.816,A -85,B 0,C 180,E1 -24992.031,E2 -24992.031} C_VEL
LIN {X 0,Y 187.525,Z 478.029,A -85,B 0,C 180,E1 -24995.654,E2 -24995.654} C_VEL
LIN {X 0,Y 186.687,Z 476.277,A -85,B 0,C 180,E1 -25000.252,E2 -25000.252} C_VEL
LIN {X 0,Y 186.938,Z 476.085,A -85,B 0,C 180,E1 -25003.871,E2 -25003.871} C_VEL
LIN {X 0,Y 187.686,Z 476.835,A -85,B 0,C 180,E1 -25006.811,E2 -25006.811} C_VEL
LIN {X 0,Y 189.482,Z 480.191,A -85,B 0,C 180,E1 -25010.929,E2 -25010.929} C_VEL
LIN {X 0,Y 191.135,Z 483.252,A -85,B 0,C 180,E1 -25013.489,E2 -25013.489} C_VEL
LIN {X 0,Y 193.65,Z 489.162,A -85,B 0,C 180,E1 -25016.704,E2 -25016.704} C_VEL
LIN {X 0,Y 195.14,Z 493.364,A -85,B 0,C 180,E1 -25018.4,E2 -25018.4} C_VEL
LIN {X 0,Y 192.267,Z 516.648,A -85,B 0,C 180,E1 -25019.264,E2 -25019.264} C_VEL
LIN {X 0,Y 189.473,Z 529.857,A -85,B 0,C 180,E1 -25020,E2 -25020} C_VEL
LIN {X 0,Y 185.841,Z 542.155,A -85,B 0,C 180,E1 -25021.042,E2 -25021.042} C_VEL
LIN {X 0,Y 181.067,Z 554.49,A -85,B 0,C 180,E1 -25022.454,E2 -25022.454} C_VEL
LIN {X 0,Y 175.557,Z 565.964,A -85,B 0,C 180,E1 -25024.248,E2 -25024.248} C_VEL
LIN {X 0,Y 169.712,Z 575.998,A -85,B 0,C 180,E1 -25026.324,E2 -25026.324} C_VEL
LIN {X 0,Y 163.569,Z 585.018,A -85,B 0,C 180,E1 -25028.782,E2 -25028.782} C_VEL
